		CASE RIFERIMENTO_POSTAZIONE_WA OF
			{Region "CENTRALE" }				
			CENTRALE :
				{Region "ROTAZIONE VERSO 180°" }					  
				IF AngoloRotazioneDestinazionePinza > 95 THEN	
					IF WorkAreaState^[iwa].Supporto.Tipologia = CAVALLETTO THEN 				
						IF (ModuleAX_Y^.Ax^.Status.ActPosition + IngombroDestinazioneY_Pos) >= (QuotaCentroPostazione - WorkAreaState^[iwa].Supporto.YDim/2) AND
							((ModuleAX_Y^.Ax^.Status.ActPosition - IngombroDestinazioneY_Neg) <= QuotaCentroPostazione) OR
							((ModuleAX_Y^.Ax^.Status.ActPosition + IngombroDestinazioneY_Pos) <= (QuotaCentroPostazione - WorkAreaState^[iwa].Supporto.YDim/2)) THEN //Se la pinza è in ingombro con il cavalletto verso SX  
								QuotaFuoriIngombro_Y_Calcolata := MIN(QuotaFuoriIngombro_Y_Calcolata,
																	QuotaCentroPostazione - 						(* Quota Y Postazione *)																									
																	WorkAreaState^[iwa].Supporto.YDim/2 -	(* Dimensione/2 del Pallet/Cassa/Cavallina *)
																	IngombroDestinazioneY_Pos -
																	OffsetSicurezza.Y.Avuoto);
								NuIngombroYCalculado180G_Depuracion := 1;											  
								IF QuotaFuoriIngombro_Y_Calcolata + IngombroDestinazioneY_Pos >= WorkFootprint^[6].Y THEN//Se supero la quota massimo dell'area di lavoro genro un allarme
									Errore := ErrCOLLISIONE_PINZA;
									ErrCollisioneDebug := 110;			 
									RETURN; 
								END_IF
								IF QuotaFuoriIngombro_Y_Calcolata - IngombroDestinazioneY_Neg <= WorkArea^[iwa].Y + INGOMBRO_RISCONTRO_BUNDLE THEN//se sono dentro all'ingombro dei supporti del bundle genero un errore
									Errore := ErrCOLLISIONE_PINZA;
									ErrCollisioneDebug := 111;			 
									RETURN; 
								END_IF			   
						ELSIF (ModuleAX_Y^.Ax^.Status.ActPosition - IngombroDestinazioneY_Neg) >= QuotaCentroPostazione THEN //Se la pinza è in ingombro con il cavalletto  
							QuotaFuoriIngombro_Y_Calcolata := MAX(QuotaFuoriIngombro_Y_Calcolata,
																QuotaCentroPostazione + 						(* Quota Y Postazione *)																									
																WorkAreaState^[iwa].Supporto.YDim/2 +	(* Dimensione/2 del Pallet/Cassa/Cavallina *)
																IngombroDestinazioneY_Neg +
																OffsetSicurezza.Y.Avuoto);
							NuIngombroYCalculado180G_Depuracion := 2;
							IF QuotaFuoriIngombro_Y_Calcolata - IngombroDestinazioneY_Neg <= WorkArea^[iwa].Y + INGOMBRO_RISCONTRO_BUNDLE THEN//se sono dentro all'ingombro dei supporti del bundle genero un errore
								Errore := ErrCOLLISIONE_PINZA;
								ErrCollisioneDebug := 112;
								RETURN;										  
							END_IF											  
							IF QuotaFuoriIngombro_Y_Calcolata + IngombroDestinazioneY_Pos >= WorkFootprint^[6].Y THEN//Se supero la quota massimo dell'area di lavoro genro un allarme
								Errore := ErrCOLLISIONE_PINZA;
								ErrCollisioneDebug := 113;			 
								RETURN; 
							END_IF
						ELSE
							QuotaFuoriIngombro_Y_Calcolata := MAX(QuotaFuoriIngombro_Y_Calcolata,                                                
																QuotaCentroPostazione + 						(* Quota Y Postazione *)				                         																					
																WorkAreaState^[iwa].Supporto.YDim/2 +	(* Dimensione/2 del Pallet/Cassa/Cavallina *)
																IngombroDestinazioneY_Neg +                                                        
																OffsetSicurezza.Y.Avuoto);  
							NuIngombroYCalculado180G_Depuracion := 3;                                                       
							IF QuotaFuoriIngombro_Y_Calcolata - IngombroDestinazioneY_Neg <= WorkArea^[iwa].Y + INGOMBRO_RISCONTRO_BUNDLE THEN//se sono dentro all'ingombro dei supporti del bundle genero un errore
								Errore := ErrCOLLISIONE_PINZA;
								ErrCollisioneDebug := 114;
								RETURN;										  
							END_IF 		
							IF QuotaFuoriIngombro_Y_Calcolata + IngombroDestinazioneY_Pos >= WorkFootprint^[6].Y THEN//Se supero la quota massimo dell'area di lavoro genro un allarme
								Errore := ErrCOLLISIONE_PINZA;
								ErrCollisioneDebug := 115;			 
								RETURN; 
							END_IF																  
						END_IF
					ELSIF WorkAreaState^[iwa].Supporto.Tipologia = BUNDLE THEN //se NELLA postazione c'è un bundle
						IF (ModuleAX_Y^.Ax^.Status.ActPosition - IngombroDestinazioneY_Neg) <= (WorkArea^[iwa].Y + INGOMBRO_RISCONTRO_BUNDLE) THEN //Se la pinza è dentro all'ingombro del bundle  
							QuotaFuoriIngombro_Y_Calcolata := MAX(QuotaFuoriIngombro_Y_Calcolata,
																	QuotaCentroPostazione + 					(* Quota Y Postazione *)																									
																	MAX(WorkAreaState^[iwa].Supporto.YDim,INGOMBRO_RISCONTRO_BUNDLE) + (* massimo tra Dimensione del bundle e dimensione riscontro *)
																	IngombroDestinazioneY_Neg +			(* Ingombro negativo pinza *)
																	OffsetSicurezza.Y.Avuoto);           (* Offset sicurezza *)
							NuIngombroYCalculado180G_Depuracion := 4;
						ELSE
							QuotaFuoriIngombro_Y_Calcolata := MAX(QuotaFuoriIngombro_Y_Calcolata,
																	QuotaCentroPostazione + 					(* Quota Y Postazione *)																									
																	MAX(WorkAreaState^[iwa].Supporto.YDim,INGOMBRO_RISCONTRO_BUNDLE) + (* massimo tra Dimensione del bundle e dimensione riscontro *)
																	IngombroDestinazioneY_Pos +			(* Ingombro negativo pinza *)
																	OffsetSicurezza.Y.Avuoto);           (* Offset sicurezza *)
							NuIngombroYCalculado180G_Depuracion := 5;
						END_IF	
					ELSE//se non c'è nulla o c'è una cassa-pianale
						QuotaFuoriIngombro_Y_Calcolata := MAX(QuotaFuoriIngombro_Y_Calcolata,ModuleAX_Y^.Ax^.Status.ActPosition,WorkSpace^.Y/2 + OffSetPosYReposo);
						IF QuotaFuoriIngombro_Y_Calcolata + IngombroDestinazioneY_Pos >= WorkFootprint^[6].Y THEN//Se supero la quota massima dell'area di lavoro genro un allarme
							Errore := ErrCOLLISIONE_PINZA;
							ErrCollisioneDebug := 116;			 
							RETURN; 
						END_IF	
						IF QuotaFuoriIngombro_Y_Calcolata - IngombroDestinazioneY_Neg <= WorkArea^[iwa].Y + INGOMBRO_RISCONTRO_BUNDLE THEN//se sono dentro all'ingombro dei supporti del bundle genero un errore
							Errore := ErrCOLLISIONE_PINZA;
							ErrCollisioneDebug := 117;			 
							RETURN; 
						END_IF	  
					END_IF
				{endregion}								   
				{Region "ROTAZIONE VERSO 0°" }
				ELSIF AngoloRotazioneDestinazionePinza < 85 THEN
					IF WorkAreaState^[iwa].Supporto.Tipologia = CAVALLETTO THEN 				
						IF (ModuleAX_Y^.Ax^.Status.ActPosition - IngombroDestinazioneY_Neg) <= (QuotaCentroPostazione + WorkAreaState^[iwa].Supporto.YDim/2) AND
						 (ModuleAX_Y^.Ax^.Status.ActPosition - IngombroDestinazioneY_Neg >= QuotaCentroPostazione) OR
						 (ModuleAX_Y^.Ax^.Status.ActPosition - IngombroDestinazioneY_Neg) >= (QuotaCentroPostazione + WorkAreaState^[iwa].Supporto.YDim/2) THEN //Se la pinza è in ingombro con il cavalletto nella zona a SX della sua metà
							QuotaFuoriIngombro_Y_Calcolata := MAX(QuotaFuoriIngombro_Y_Calcolata,
																QuotaCentroPostazione + 						(* Quota Y Postazione *)																									
																WorkAreaState^[iwa].Supporto.YDim/2 +	(* Dimensione/2 del Pallet/Cassa/Cavallina *)
																IngombroDestinazioneY_Neg +
																OffsetSicurezza.Y.Avuoto);
							NuIngombroYCalculado0G_Depuracion := 1;
							IF QuotaFuoriIngombro_Y_Calcolata + IngombroDestinazioneY_Pos >= WorkFootprint^[6].Y THEN//Se supero la quota massimo dell'area di lavoro genro un allarme
								Errore := ErrCOLLISIONE_PINZA;
								ErrCollisioneDebug := 118;			 
								RETURN; 
							END_IF 
						ELSIF ((ModuleAX_Y^.Ax^.Status.ActPosition + IngombroDestinazioneY_Pos) >= (QuotaCentroPostazione - WorkAreaState^[iwa].Supporto.YDim/2) AND 
							(ModuleAX_Y^.Ax^.Status.ActPosition + IngombroDestinazioneY_Pos) <= (QuotaCentroPostazione)) OR
							(ModuleAX_Y^.Ax^.Status.ActPosition + IngombroDestinazioneY_Pos) <= (QuotaCentroPostazione)THEN //Se la pinza è in ingombro con il cavalletto con pinza dentro all'ingombro nella parte SX 
								QuotaFuoriIngombro_Y_Calcolata := MIN(QuotaFuoriIngombro_Y_Calcolata,
																	QuotaCentroPostazione - 						(* Quota Y Postazione *)																									
																	WorkAreaState^[iwa].Supporto.YDim/2 -	(* Dimensione/2 del Pallet/Cassa/Cavallina *)
																	IngombroDestinazioneY_Pos -
																	OffsetSicurezza.Y.Avuoto);
								NuIngombroYCalculado0G_Depuracion := 2;
								IF QuotaFuoriIngombro_Y_Calcolata - IngombroDestinazioneY_Neg <= WorkArea^[iwa].Y + INGOMBRO_RISCONTRO_BUNDLE THEN//se sono dentro all'ingombro dei supporti del bundle genero un errore
									Errore := ErrCOLLISIONE_PINZA;
									ErrCollisioneDebug := 119;
									RETURN;										  
								END_IF 							
						ELSE
							QuotaFuoriIngombro_Y_Calcolata := MAX(QuotaFuoriIngombro_Y_Calcolata,
																QuotaCentroPostazione + 						(* Quota Y Postazione *)																									
																WorkAreaState^[iwa].Supporto.YDim/2 +	(* Dimensione/2 del Pallet/Cassa/Cavallina *)
																IngombroDestinazioneY_Neg +				(* Ingombro positivo pinza *)
																OffsetSicurezza.Y.Avuoto);				(* Offset sicurezza *)
							NuIngombroYCalculado0G_Depuracion := 3;
							IF QuotaFuoriIngombro_Y_Calcolata - IngombroDestinazioneY_Neg <= WorkArea^[iwa].Y + INGOMBRO_RISCONTRO_BUNDLE THEN//se sono dentro all'ingombro dei supporti del bundle genero un errore
								Errore := ErrCOLLISIONE_PINZA;
								ErrCollisioneDebug := 120;
								RETURN;										  
							END_IF 
							IF QuotaFuoriIngombro_Y_Calcolata + IngombroDestinazioneY_Pos >= WorkFootprint^[6].Y THEN//Se supero la quota massimo dell'area di lavoro genro un allarme
								Errore := ErrCOLLISIONE_PINZA;
								ErrCollisioneDebug := 121;			 
								RETURN; 
							END_IF
						END_IF
					ELSIF WorkAreaState^[iwa].Supporto.Tipologia = BUNDLE THEN //se NELLA postazione c'è un bundle
						IF (ModuleAX_Y^.Ax^.Status.ActPosition - IngombroDestinazioneY_Neg) <= (QuotaCentroPostazione + INGOMBRO_RISCONTRO_BUNDLE) THEN //Se la pinza è dentro all'ingombro del bundle  
							QuotaFuoriIngombro_Y_Calcolata := MAX(QuotaFuoriIngombro_Y_Calcolata,
																	QuotaCentroPostazione + 					(* Quota Y Postazione *)																									
																	MAX(WorkAreaState^[iwa].Supporto.YDim,INGOMBRO_RISCONTRO_BUNDLE) + (* massimo tra Dimensione del bundle e dimensione riscontro *)
																	IngombroDestinazioneY_Neg +			(* Ingombro negativo pinza *)
																	OffsetSicurezza.Y.Avuoto);           (* Offset sicurezza *)
							NuIngombroYCalculado0G_Depuracion := 4;
							IF QuotaFuoriIngombro_Y_Calcolata - IngombroDestinazioneY_Neg <= WorkArea^[iwa].Y + INGOMBRO_RISCONTRO_BUNDLE THEN//se sono dentro all'ingombro dei supporti del bundle genero un errore
								Errore := ErrCOLLISIONE_PINZA;
								ErrCollisioneDebug := 122;
								RETURN;										  
							END_IF 
							IF QuotaFuoriIngombro_Y_Calcolata + IngombroDestinazioneY_Pos >= WorkFootprint^[6].Y THEN//Se supero la quota massimo dell'area di lavoro genro un allarme
								Errore := ErrCOLLISIONE_PINZA;
								ErrCollisioneDebug := 123;			 
								RETURN; 
							END_IF												  
						ELSE
							QuotaFuoriIngombro_Y_Calcolata := MAX(QuotaFuoriIngombro_Y_Calcolata,
																	QuotaCentroPostazione + 					(* Quota Y Postazione *)																									
																	MAX(WorkAreaState^[iwa].Supporto.YDim,INGOMBRO_RISCONTRO_BUNDLE) + (* massimo tra Dimensione del bundle e dimensione riscontro *)
																	IngombroDestinazioneY_Pos +			(* Ingombro negativo pinza *)
																	OffsetSicurezza.Y.Avuoto);           (* Offset sicurezza *)
							NuIngombroYCalculado0G_Depuracion := 5;
							IF QuotaFuoriIngombro_Y_Calcolata - IngombroDestinazioneY_Neg <= QuotaCentroPostazione + INGOMBRO_RISCONTRO_BUNDLE THEN//se sono dentro all'ingombro dei supporti del bundle genero un errore
								Errore := ErrCOLLISIONE_PINZA;
								ErrCollisioneDebug := 124;
								RETURN;										  
							END_IF 
							IF QuotaFuoriIngombro_Y_Calcolata + IngombroDestinazioneY_Pos >= WorkFootprint^[6].Y THEN//Se supero la quota massimo dell'area di lavoro genro un allarme
								Errore := ErrCOLLISIONE_PINZA;
								ErrCollisioneDebug := 125;			 
								RETURN; 
							END_IF												  
						END_IF	
					ELSE//se non c'è nulla o c'è una cassa-pianale
						QuotaFuoriIngombro_Y_Calcolata := MAX(QuotaFuoriIngombro_Y_Calcolata,ModuleAX_Y^.Ax^.Status.ActPosition,WorkSpace^.Y/2 +OffSetPosYReposo);
						IF QuotaFuoriIngombro_Y_Calcolata + IngombroDestinazioneY_Pos >= WorkFootprint^[6].Y THEN//Se supero la quota massima dell'area di lavoro genro un allarme
							Errore := ErrCOLLISIONE_PINZA;
							ErrCollisioneDebug := 126;			 
							RETURN; 
						END_IF	
						IF QuotaFuoriIngombro_Y_Calcolata - IngombroDestinazioneY_Neg <= WorkArea^[iwa].Y + INGOMBRO_RISCONTRO_BUNDLE THEN//se sono dentro all'ingombro dei supporti del bundle genero un errore
							Errore := ErrCOLLISIONE_PINZA;
							ErrCollisioneDebug := 127;			 
							RETURN; 
						END_IF	  
					END_IF 	
				{endregion}								   
				{Region "ROTAZIONE 90°" }
				ELSE	
					IF WorkAreaState^[iwa].Supporto.Tipologia = CAVALLETTO THEN 				
						IF (ModuleAX_Y^.Ax^.Status.ActPosition - IngombroDestinazioneY_Neg) <= (QuotaCentroPostazione + WorkAreaState^[iwa].Supporto.YDim/2) AND
							(ModuleAX_Y^.Ax^.Status.ActPosition - IngombroDestinazioneY_Neg >= QuotaCentroPostazione) THEN //Se la pinza è in ingombro con il cavalletto nella zona a DX della sua metà
							QuotaFuoriIngombro_Y_Calcolata := MAX(QuotaFuoriIngombro_Y_Calcolata,
																QuotaCentroPostazione + 						(* Quota Y Postazione *)																									
																WorkAreaState^[iwa].Supporto.YDim/2 +	(* Dimensione/2 del Pallet/Cassa/Cavallina *)
																IngombroDestinazioneY_Neg +
																OffsetSicurezza.Y.Avuoto);
						NuIngombroYCalculado90G_Depuracion := 1 ;
							IF QuotaFuoriIngombro_Y_Calcolata + IngombroDestinazioneY_Pos >= WorkFootprint^[6].Y THEN//Se supero la quota massimo dell'area di lavoro genro un allarme
								Errore := ErrCOLLISIONE_PINZA;
								ErrCollisioneDebug := 128;			 
								RETURN; 
							END_IF 
						ELSIF (ModuleAX_Y^.Ax^.Status.ActPosition + IngombroDestinazioneY_Pos) >= (QuotaCentroPostazione - WorkAreaState^[iwa].Supporto.YDim/2) AND 
							(ModuleAX_Y^.Ax^.Status.ActPosition + IngombroDestinazioneY_Pos) <= (QuotaCentroPostazione) THEN //Se la pinza è in ingombro con il cavalletto con pinza dentro all'ingombro nella parte SX 
								QuotaFuoriIngombro_Y_Calcolata := MIN(QuotaFuoriIngombro_Y_Calcolata,
																	QuotaCentroPostazione - 						(* Quota Y Postazione *)																									
																	WorkAreaState^[iwa].Supporto.YDim/2 -	(* Dimensione/2 del Pallet/Cassa/Cavallina *)
																	IngombroDestinazioneY_Pos -
																	OffsetSicurezza.Y.Avuoto);
							NuIngombroYCalculado90G_Depuracion := 2 ;
								IF QuotaFuoriIngombro_Y_Calcolata - IngombroDestinazioneY_Neg <= WorkArea^[iwa].Y + INGOMBRO_RISCONTRO_BUNDLE THEN//se sono dentro all'ingombro dei supporti del bundle genero un errore
									Errore := ErrCOLLISIONE_PINZA;
									ErrCollisioneDebug := 129;
									RETURN;										  
								END_IF 							
						ELSE
							QuotaFuoriIngombro_Y_Calcolata := MAX(QuotaFuoriIngombro_Y_Calcolata,
																QuotaCentroPostazione + 						(* Quota Y Postazione *)																									
																WorkAreaState^[iwa].Supporto.YDim/2 +	(* Dimensione/2 del Pallet/Cassa/Cavallina *)
																IngombroDestinazioneY_Neg +				(* Ingombro positivo pinza *)
																OffsetSicurezza.Y.Avuoto);				(* Offset sicurezza *)
							NuIngombroYCalculado90G_Depuracion := 3 ;
							IF QuotaFuoriIngombro_Y_Calcolata - IngombroDestinazioneY_Neg <= WorkArea^[iwa].Y + INGOMBRO_RISCONTRO_BUNDLE THEN//se sono dentro all'ingombro dei supporti del bundle genero un errore
								Errore := ErrCOLLISIONE_PINZA;
								ErrCollisioneDebug := 130;
								RETURN;										  
							END_IF 
							IF QuotaFuoriIngombro_Y_Calcolata + IngombroDestinazioneY_Pos >= WorkFootprint^[6].Y THEN//Se supero la quota massimo dell'area di lavoro genro un allarme
								Errore := ErrCOLLISIONE_PINZA;
								ErrCollisioneDebug := 131;			 
								RETURN; 
							END_IF
						END_IF
					ELSIF WorkAreaState^[iwa].Supporto.Tipologia = BUNDLE THEN //se NELLA postazione c'è un bundle
						IF (ModuleAX_Y^.Ax^.Status.ActPosition - IngombroDestinazioneY_Neg) <= (WorkArea^[iwa].Y + INGOMBRO_RISCONTRO_BUNDLE) THEN //Se la pinza è dentro all'ingombro del bundle  
							QuotaFuoriIngombro_Y_Calcolata := MAX(QuotaFuoriIngombro_Y_Calcolata,
																	QuotaCentroPostazione + 					(* Quota Y Postazione *)																									
																	MAX(WorkAreaState^[iwa].Supporto.YDim,INGOMBRO_RISCONTRO_BUNDLE) + (* massimo tra Dimensione del bundle e dimensione riscontro *)
																	IngombroDestinazioneY_Neg +			(* Ingombro negativo pinza *)
																	OffsetSicurezza.Y.Avuoto);           (* Offset sicurezza *)
							NuIngombroYCalculado90G_Depuracion := 4 ;
							IF QuotaFuoriIngombro_Y_Calcolata - IngombroDestinazioneY_Neg <= WorkArea^[iwa].Y + INGOMBRO_RISCONTRO_BUNDLE THEN//se sono dentro all'ingombro dei supporti del bundle genero un errore
								Errore := ErrCOLLISIONE_PINZA;
								ErrCollisioneDebug := 132;
								RETURN;										  
							END_IF 
							IF QuotaFuoriIngombro_Y_Calcolata + IngombroDestinazioneY_Pos >= WorkFootprint^[6].Y THEN//Se supero la quota massimo dell'area di lavoro genro un allarme
								Errore := ErrCOLLISIONE_PINZA;
								ErrCollisioneDebug := 133;			 
								RETURN; 
							END_IF												  
						ELSE
							QuotaFuoriIngombro_Y_Calcolata := MAX(QuotaFuoriIngombro_Y_Calcolata,
																	QuotaCentroPostazione + 					(* Quota Y Postazione *)																									
																	MAX(WorkAreaState^[iwa].Supporto.YDim,INGOMBRO_RISCONTRO_BUNDLE) + (* massimo tra Dimensione del bundle e dimensione riscontro *)
																	IngombroDestinazioneY_Pos +			(* Ingombro negativo pinza *)
																	OffsetSicurezza.Y.Avuoto);           (* Offset sicurezza *)
							NuIngombroYCalculado90G_Depuracion := 5 ;
							IF QuotaFuoriIngombro_Y_Calcolata - IngombroDestinazioneY_Neg <= WorkArea^[iwa].Y + INGOMBRO_RISCONTRO_BUNDLE THEN//se sono dentro all'ingombro dei supporti del bundle genero un errore
								Errore := ErrCOLLISIONE_PINZA;
								ErrCollisioneDebug := 134;
								RETURN;										  
							END_IF 
							IF QuotaFuoriIngombro_Y_Calcolata + IngombroDestinazioneY_Pos >= WorkFootprint^[6].Y THEN//Se supero la quota massimo dell'area di lavoro genro un allarme
								Errore := ErrCOLLISIONE_PINZA;
								ErrCollisioneDebug := 135;			 
								RETURN; 
							END_IF												  
						END_IF	
					ELSE//se non c'è nulla o c'è una cassa-pianale
						QuotaFuoriIngombro_Y_Calcolata := MAX(QuotaFuoriIngombro_Y_Calcolata,ModuleAX_Y^.Ax^.Status.ActPosition,WorkSpace^.Y/2+ OffSetPosYReposo);
						IF QuotaFuoriIngombro_Y_Calcolata + IngombroDestinazioneY_Pos >= WorkFootprint^[6].Y THEN//Se supero la quota massima dell'area di lavoro genro un allarme
							Errore := ErrCOLLISIONE_PINZA;
							ErrCollisioneDebug := 136;			 
							RETURN; 
						END_IF	
						IF QuotaFuoriIngombro_Y_Calcolata - IngombroDestinazioneY_Neg <= WorkArea^[iwa].Y + INGOMBRO_RISCONTRO_BUNDLE THEN//se sono dentro all'ingombro dei supporti del bundle genero un errore
							Errore := ErrCOLLISIONE_PINZA;
							ErrCollisioneDebug := 137;			 
							RETURN; 
						END_IF	  
					END_IF
				END_IF
				{endregion}				   
			{endregion}
		
		ELSE
			;//Errore.Code := ErrWAM_FTC_PostazioneNONDefinita;
		END_CASE
	{endregion}	
	{region " Pallettizzatore SX "}	
	PALLETTIZZATORE_SX:
		CASE RIFERIMENTO_POSTAZIONE_WA OF
		{Region "CENTRALE" }				
			CENTRALE :
				{Region "ROTAZIONE VERSO 180°" }					  
				IF AngoloRotazioneDestinazionePinza > 95 THEN
					//Modificacar aqui para salir <cavaleta	
					IF WorkAreaState^[iwa].Supporto.Tipologia = CAVALLETTO  (*Añadido*)OR WorkAreaState^[PosRobot].Supporto.Tipologia = CAVALLETTO 
							OR (WorkAreaState^[Mission^.PPlace].Supporto.Tipologia = CAVALLETTO	AND WorkAreaManager^.State = 	WAMANAGER_CICLO_DEPOSITO_LASTRA_WA_RUN)	THEN 				
						IF (ModuleAX_Y^.Ax^.Status.ActPosition + IngombroDestinazioneY_Pos) >= (QuotaCentroPostazione - WorkAreaState^[iwa].Supporto.YDim/2) AND
							((ModuleAX_Y^.Ax^.Status.ActPosition - IngombroDestinazioneY_Neg) <= QuotaCentroPostazione) OR
							((ModuleAX_Y^.Ax^.Status.ActPosition + IngombroDestinazioneY_Pos) <= (QuotaCentroPostazione - WorkAreaState^[iwa].Supporto.YDim/2)) OR
							 	( (WorkAreaState^[PosRobot].Supporto.Tipologia = CAVALLETTO OR WorkAreaState^[Mission^.PPlace].Supporto.Tipologia = CAVALLETTO ) AND ModuleAX_Y^.Ax^.Status.ActPosition + IngombroDestinazioneY_Pos < WorkFootprint^[6].Y )THEN //Se la pinza è in ingombro con il cavalletto verso SX  
							 	IF WorkAreaState^[PosRobot].Supporto.Tipologia = CAVALLETTO OR  
											WorkAreaState^[Mission^.PPlace].Supporto.Tipologia = CAVALLETTO THEN
									IF WorkAreaState^[Mission^.PPlace].Supporto.Tipologia = CAVALLETTO AND WorkAreaManager^.State = 	WAMANAGER_CICLO_DEPOSITO_LASTRA_WA_RUN  THEN
											QuotaFuoriIngombro_Y_Calcolata := 
													   //%%%%%%%%%%%%%%%%modificado 18-7-2025
																			MAX(QuotaFuoriIngombro_Y_Calcolata,
																			QuotaCentroPostazionePiking + 						(* Quota Y Postazione *)																									
																			WorkAreaState^[Mission^.PPlace].Supporto.YDim/2 (*-	        (* Dimensione/2 del Pallet/Cassa/Cavallina *)
																			IngombroDestinazioneY_Pos - *) 
																			+ Max (OffsetSicurezza.Y.Avuoto ,Dimensioni_Pinza.Spessore)           )  ;
									NuIngombroYCalculado180G_Depuracion := 6;
									ELSE
										IF Mission^.PPick = PosRobot AND( Mission^.JPick <> Mission^.JPlace OR ModuleAX_J^.Ax^.Status.ActPosition < 85) THEN
														   
											IF 	Mission^.JPick < 85 THEN
											QuotaFuoriIngombro_Y_Calcolata := 
											 //%%%%%%%%%%%%%%%%modificado 18-7-2025
																			MAX(QuotaFuoriIngombro_Y_Calcolata,
																			QuotaCentroPostazioneIni - 						(* Quota Y Postazione *)																									
																			WorkAreaState^[Mission^.PPick].Supporto.YDim/2 (*-	        (* Dimensione/2 del Pallet/Cassa/Cavallina *)
																			IngombroDestinazioneY_Pos - *) 
																			- OffsetSicurezza.Y.Avuoto )  ;	
											NuIngombroYCalculado180G_Depuracion := 7;	   
	   										ELSE
											QuotaFuoriIngombro_Y_Calcolata := 
											 //%%%%%%%%%%%%%%%%modificado 18-7-2025
																			MAX(QuotaFuoriIngombro_Y_Calcolata,
																			QuotaCentroPostazioneIni + 						(* Quota Y Postazione *)																									
																			WorkAreaState^[Mission^.PPick].Supporto.YDim/2 (*-	        (* Dimensione/2 del Pallet/Cassa/Cavallina *)
																			IngombroDestinazioneY_Pos - *) 
																			+ OffsetSicurezza.Y.Avuoto )  ;	
											NuIngombroYCalculado180G_Depuracion := 8;	   				   
											END_IF	
										// Añadido 	29 -7-2025__________________________________________			   
										ELSIF   PosRobot <> 0 AND   WorkAreaState^[PosRobot].Supporto.Tipologia = CAVALLETTO  AND ModuleAX_J^.Ax^.Status.ActPosition > 95      THEN 
											QuotaFuoriIngombro_Y_Calcolata := 
											 //%%%%%%%%%%%%%%%%modificado 18-7-2025
																			MAX(QuotaFuoriIngombro_Y_Calcolata,
																			QuotaCentroPostazioneIni  + 						(* Quota Y Postazione *)	
																			//	WorkAreaState^[Mission^.PPick].Supporto.YDim/2				
																			WorkAreaState^[PosRobot].Supporto.YDim /2 (*-	        (* Dimensione/2 del Pallet/Cassa/Cavallina *)
																			
																			IngombroDestinazioneY_Pos - *) 
																			+ OffsetSicurezza.Y.Avuoto +INGOMBRO_RISCONTRO_FRAME )  ;
										NuIngombroYCalculado180G_Depuracion := 9;			   			   
		   								// Añadido 	29 -7-2025_________________________________________________
										ELSIF PosRobot <> 0 AND  WorkAreaState^[PosRobot].Supporto.Tipologia = CAVALLETTO  AND ModuleAX_J^.Ax^.Status.ActPosition < 95    THEN 
											
																			
																			IF 	WorkAreaState^[Mission^.PPick].Supporto.Tipologia = BUNDLE THEN
																				Soporte := WorkAreaState^[Mission^.PPick].Supporto.YDim;	
																			ELSIF WorkAreaState^[Mission^.PPick].Supporto.Tipologia = CAVALLETTO THEN
																				Soporte := WorkAreaState^[Mission^.PPick].Supporto.YDim /2;	   
																			END_IF		   
																			QuotaFuoriIngombro_Y_Calcolata := 
																			 //%%%%%%%%%%%%%%%%modificado 18-7-2025														  
																			//Modificacion Pasillo Trabajo Caballete
																			MAX(QuotaFuoriIngombro_Y_Calcolata,
																			QuotaCentroPostazione  + 					(* Quota Y Postazione *)	
																			Soporte
																			+ MAX( OffsetSicurezza.Y.Avuoto , Dimensioni_Pinza.Spessore))  ;
										NuIngombroYCalculado180G_Depuracion := 10;		   			   
		   								// Añadido 	2 -9-2025_________________________________________________
										ELSIF (( WorkAreaState^[Mission^.PPick].Supporto.Tipologia = CAVALLETTO  AND NuPosGuiroPiking = PosRobot) OR ( PosRobot <> 0 AND WorkAreaState^[PosRobot].Supporto.Tipologia <> CAVALLETTO))  AND PosicionJActual = 90     THEN 
											QuotaFuoriIngombro_Y_Calcolata := 
											 //%%%%%%%%%%%%%%%%modificado 2-9-2025
																			MAX(QuotaFuoriIngombro_Y_Calcolata,
																			QuotaCentroPostazione  + 						(* Quota Y Postazione *)	
																			//	WorkAreaState^[Mission^.PPick].Supporto.YDim/2				
																			WorkAreaState^[Mission^.PPick].Supporto.YDim /2 + Dimensioni_Pinza.Spessore(*-	        (* Dimensione/2 del Pallet/Cassa/Cavallina *)
																			
																			IngombroDestinazioneY_Pos - *) 
																			(*+ OffsetSicurezza.Y.Avuoto *)+ INGOMBRO_RISCONTRO_FRAME)  ;	
										NuIngombroYCalculado180G_Depuracion := 11;		
										// Añadido 	4 -9-2025_________________________________________________
										ELSIF  WorkAreaState^[Mission^.PPick].Supporto.Tipologia = BUNDLE  AND  PosRobot = 0    THEN 
											QuotaFuoriIngombro_Y_Calcolata := 
											 //%%%%%%%%%%%%%%%%modificado 2-9-2025
																			MAX(QuotaFuoriIngombro_Y_Calcolata,
																			QuotaCentroPostazione  + 						(* Quota Y Postazione *)	
																			//	WorkAreaState^[Mission^.PPick].Supporto.YDim/2				
																			WorkAreaState^[Mission^.PPick].Supporto.YDim /2 (*-	        (* Dimensione/2 del Pallet/Cassa/Cavallina *)
																			
																			IngombroDestinazioneY_Pos - *) 
																			+ OffsetSicurezza.Y.Avuoto )  ;		
										NuIngombroYCalculado180G_Depuracion := 12;	   		   			
										END_IF
										 
									END_IF
								ELSE
										IF 	WorkAreaState^[Mission^.PPlace].Supporto.Tipologia = CAVALLETTO	 THEN
  											QuotaFuoriIngombro_Y_Calcolata := 
											   //%%%%%%%%%%%%%%%%modificado 18-7-2025
											   						MAX(QuotaFuoriIngombro_Y_Calcolata,
																	QuotaCentroPostazione + 						(* Quota Y Postazione *)																									
																	WorkAreaState^[iwa].Supporto.YDim/2 (*-	        (* Dimensione/2 del Pallet/Cassa/Cavallina *)
																	IngombroDestinazioneY_Pos - *) 
																	+ OffsetSicurezza.Y.Avuoto + INGOMBRO_RISCONTRO_FRAME )  ;
										NuIngombroYCalculado180G_Depuracion := 13;
										ELSIF WorkAreaState^[Mission^.PPlace].Supporto.Tipologia = BUNDLE    THEN  	
											QuotaFuoriIngombro_Y_Calcolata := 
											   //%%%%%%%%%%%%%%%%modificado 18-7-2025
											   						MAX(QuotaFuoriIngombro_Y_Calcolata,
																	QuotaCentroPostazione + 						(* Quota Y Postazione *)																									
																	WorkAreaState^[iwa].Supporto.YDim /2  (*-	        (* Dimensione/2 del Pallet/Cassa/Cavallina *)
																	IngombroDestinazioneY_Pos - *) 
																	+MAX(Dimensioni_Pinza.Spessore ,OffsetSicurezza.Y.Avuoto ))+ INGOMBRO_RISCONTRO_FRAME   ;
										NuIngombroYCalculado180G_Depuracion := 14;
											ELSIF WorkAreaState^[Mission^.PPick].Supporto.Tipologia = CAVALLETTO    THEN  	
											QuotaFuoriIngombro_Y_Calcolata := 
											   //%%%%%%%%%%%%%%%%modificado 18-7-2025
											   						MAX(QuotaFuoriIngombro_Y_Calcolata,
																	QuotaCentroPostazione + 						(* Quota Y Postazione *)																									
																	WorkAreaState^[iwa].Supporto.YDim /2 (*-	        (* Dimensione/2 del Pallet/Cassa/Cavallina *)
																	IngombroDestinazioneY_Pos - *) 
																	+ max ( Dimensioni_Pinza.Spessore ,  OffsetSicurezza.Y.Avuoto )+ INGOMBRO_RISCONTRO_FRAME )  ;	
										NuIngombroYCalculado180G_Depuracion := 15;							
										END_IF 
					  
			   						
								END_IF 		   
										(*	QuotaFuoriIngombro_Y_Calcolata := 
											   //%%%%%%%%%%%%%%%%modificado 18-7-2025
											   						MAX(QuotaFuoriIngombro_Y_Calcolata,
																	QuotaCentroPostazione + 						(* Quota Y Postazione *)																									
																	WorkAreaState^[iwa].Supporto.YDim/2 (*-	        (* Dimensione/2 del Pallet/Cassa/Cavallina *)
																	IngombroDestinazioneY_Pos - *) 
																	+ OffsetSicurezza.Y.Avuoto )  ;
																(*	MIN(QuotaFuoriIngombro_Y_Calcolata,
																	QuotaCentroPostazione - 						(* Quota Y Postazione *)																									
																	WorkAreaState^[iwa].Supporto.YDim/2 -	(* Dimensione/2 del Pallet/Cassa/Cavallina *)
																	IngombroDestinazioneY_Pos -
																	OffsetSicurezza.Y.Avuoto);*)
																			  *)
								IF QuotaFuoriIngombro_Y_Calcolata (*+ IngombroDestinazioneY_Pos*) >= WorkFootprint^[6].Y THEN//Se supero la quota massimo dell'area di lavoro genro un allarme
									Errore := ErrCOLLISIONE_PINZA;
									ErrCollisioneDebug := 10;			 
									RETURN; 
								END_IF
								IF QuotaFuoriIngombro_Y_Calcolata - IngombroDestinazioneY_Neg <= WorkArea^[iwa].Y + INGOMBRO_RISCONTRO_BUNDLE THEN//se sono dentro all'ingombro dei supporti del bundle genero un errore
									Errore := ErrCOLLISIONE_PINZA;
									ErrCollisioneDebug := 11;			 
									RETURN; 
								END_IF			   
						ELSIF (ModuleAX_Y^.Ax^.Status.ActPosition - IngombroDestinazioneY_Neg) >= QuotaCentroPostazione THEN //Se la pinza è in ingombro con il cavalletto  
							QuotaFuoriIngombro_Y_Calcolata := MAX(QuotaFuoriIngombro_Y_Calcolata,
																QuotaCentroPostazione + 						(* Quota Y Postazione *)																									
																WorkAreaState^[iwa].Supporto.YDim/2 +	(* Dimensione/2 del Pallet/Cassa/Cavallina *)
																IngombroDestinazioneY_Neg + INGOMBRO_RISCONTRO_FRAME(*+
																OffsetSicurezza.Y.Avuoto*));
							NuIngombroYCalculado180G_Depuracion := 16;
							IF QuotaFuoriIngombro_Y_Calcolata - IngombroDestinazioneY_Neg <= WorkArea^[iwa].Y + INGOMBRO_RISCONTRO_BUNDLE THEN//se sono dentro all'ingombro dei supporti del bundle genero un errore
								Errore := ErrCOLLISIONE_PINZA;
								ErrCollisioneDebug := 12;
								RETURN;										  
							END_IF											  
							IF QuotaFuoriIngombro_Y_Calcolata + IngombroDestinazioneY_Pos /2(*Puesto Para Probar*)  >= WorkFootprint^[6].Y THEN//Se supero la quota massimo dell'area di lavoro genro un allarme
								Errore := ErrCOLLISIONE_PINZA;
								ErrCollisioneDebug := 13;			 
								RETURN; 
							END_IF
						ELSE
							QuotaFuoriIngombro_Y_Calcolata := MAX(QuotaFuoriIngombro_Y_Calcolata,                                                
																QuotaCentroPostazione + 						(* Quota Y Postazione *)				                         																					
																WorkAreaState^[iwa].Supporto.YDim/2 +	(* Dimensione/2 del Pallet/Cassa/Cavallina *)
																(*IngombroDestinazioneY_Neg + *) //+++++++++                                                      
																OffsetSicurezza.Y.Avuoto);  
							NuIngombroYCalculado180G_Depuracion := 17;                                                       
							IF QuotaFuoriIngombro_Y_Calcolata - IngombroDestinazioneY_Neg <= WorkArea^[iwa].Y + INGOMBRO_RISCONTRO_BUNDLE THEN//se sono dentro all'ingombro dei supporti del bundle genero un errore
								Errore := ErrCOLLISIONE_PINZA;
								ErrCollisioneDebug := 14;
								RETURN;										  
							END_IF 		
							IF QuotaFuoriIngombro_Y_Calcolata + IngombroDestinazioneY_Pos >= WorkFootprint^[6].Y THEN//Se supero la quota massimo dell'area di lavoro genro un allarme
								Errore := ErrCOLLISIONE_PINZA;
								ErrCollisioneDebug := 15;			 
								RETURN; 
							END_IF																  
						END_IF
					ELSIF WorkAreaState^[iwa].Supporto.Tipologia = BUNDLE THEN //se NELLA postazione c'è un bundle
						IF (ModuleAX_Y^.Ax^.Status.ActPosition - IngombroDestinazioneY_Neg) <= (WorkArea^[iwa].Y + INGOMBRO_RISCONTRO_BUNDLE) THEN //Se la pinza è dentro all'ingombro del bundle  
							QuotaFuoriIngombro_Y_Calcolata := MAX(QuotaFuoriIngombro_Y_Calcolata,
																	QuotaCentroPostazione + 					(* Quota Y Postazione *)																									
																	MAX(WorkAreaState^[iwa].Supporto.YDim,INGOMBRO_RISCONTRO_BUNDLE) + (* massimo tra Dimensione del bundle e dimensione riscontro *)
																	MAX (IngombroDestinazioneY_Neg ,			(* Ingombro negativo pinza *)
																	OffsetSicurezza.Y.Avuoto));           (* Offset sicurezza *)
						NuIngombroYCalculado180G_Depuracion := 18; 
						ELSE
							QuotaFuoriIngombro_Y_Calcolata := MAX(QuotaFuoriIngombro_Y_Calcolata,
																	QuotaCentroPostazione + 					(* Quota Y Postazione *)																									
																	MAX(WorkAreaState^[iwa].Supporto.YDim,INGOMBRO_RISCONTRO_BUNDLE) + (* massimo tra Dimensione del bundle e dimensione riscontro *)
																	MAX (IngombroDestinazioneY_Pos  ,			(* Ingombro negativo pinza *)
																	OffsetSicurezza.Y.Avuoto, Dimensioni_Pinza.Spessore) +INGOMBRO_RISCONTRO_BUNDLE);           (* Offset sicurezza *)
						NuIngombroYCalculado180G_Depuracion := 19; 
						END_IF	
					ELSE//se non c'è nulla o c'è una cassa-pianale
						QuotaFuoriIngombro_Y_Calcolata := MAX(QuotaFuoriIngombro_Y_Calcolata,ModuleAX_Y^.Ax^.Status.ActPosition,WorkSpace^.Y/2 + OffSetPosYReposo);
						IF QuotaFuoriIngombro_Y_Calcolata + IngombroDestinazioneY_Pos >= WorkFootprint^[6].Y THEN//Se supero la quota massima dell'area di lavoro genro un allarme
							Errore := ErrCOLLISIONE_PINZA;
							ErrCollisioneDebug := 16;			 
							RETURN; 
						END_IF	
						IF QuotaFuoriIngombro_Y_Calcolata - IngombroDestinazioneY_Neg <= WorkArea^[iwa].Y + INGOMBRO_RISCONTRO_BUNDLE THEN//se sono dentro all'ingombro dei supporti del bundle genero un errore
							Errore := ErrCOLLISIONE_PINZA;
							ErrCollisioneDebug := 17;			 
							RETURN; 
						END_IF	  
					END_IF
				{endregion}								   
				{Region "ROTAZIONE VERSO 0°" }
				ELSIF AngoloRotazioneDestinazionePinza < 85 THEN
					IF WorkAreaState^[iwa].Supporto.Tipologia = CAVALLETTO THEN 				
						IF (ModuleAX_Y^.Ax^.Status.ActPosition - IngombroDestinazioneY_Neg) <= (QuotaCentroPostazione + WorkAreaState^[iwa].Supporto.YDim/2) AND
							(ModuleAX_Y^.Ax^.Status.ActPosition - IngombroDestinazioneY_Neg >= QuotaCentroPostazione) THEN //Se la pinza è in ingombro con il cavalletto nella zona a DX della sua metà
							QuotaFuoriIngombro_Y_Calcolata := MAX(QuotaFuoriIngombro_Y_Calcolata,
																QuotaCentroPostazione - 						(* Quota Y Postazione *)																									
																WorkAreaState^[iwa].Supporto.YDim/2 -	(* Dimensione/2 del Pallet/Cassa/Cavallina *)
																IngombroDestinazioneY_Neg  -
																OffsetSicurezza.Y.Avuoto );
						   NuIngombroYCalculado0G_Depuracion := 6;	
							(*												   
							QuotaFuoriIngombro_Y_Calcolata := MAX(QuotaFuoriIngombro_Y_Calcolata,
																QuotaCentroPostazione + 						(* Quota Y Postazione *)																									
																WorkAreaState^[iwa].Supporto.YDim/2 +	(* Dimensione/2 del Pallet/Cassa/Cavallina *)
																IngombroDestinazioneY_Neg +
																OffsetSicurezza.Y.Avuoto);												   
								*)
							IF QuotaFuoriIngombro_Y_Calcolata + IngombroDestinazioneY_Pos >= WorkFootprint^[6].Y THEN//Se supero la quota massimo dell'area di lavoro genro un allarme
								Errore := ErrCOLLISIONE_PINZA;
								ErrCollisioneDebug := 18;			 
								RETURN; 
							END_IF 
						ELSIF (ModuleAX_Y^.Ax^.Status.ActPosition + IngombroDestinazioneY_Pos) >= (QuotaCentroPostazione - WorkAreaState^[iwa].Supporto.YDim/2) AND 
							(ModuleAX_Y^.Ax^.Status.ActPosition + IngombroDestinazioneY_Pos <= QuotaCentroPostazione) THEN //Se la pinza è in ingombro con il cavalletto con pinza dentro all'ingombro nella parte SX 
								QuotaFuoriIngombro_Y_Calcolata := //MIN(QuotaFuoriIngombro_Y_Calcolata,
												   				   MAX(QuotaFuoriIngombro_Y_Calcolata,
																	QuotaCentroPostazione - 						(* Quota Y Postazione *)																									
																	WorkAreaState^[iwa].Supporto.YDim/2 -	(* Dimensione/2 del Pallet/Cassa/Cavallina *)
																	MAX( IngombroDestinazioneY_Pos ,
																	OffsetSicurezza.Y.Avuoto));
							   NuIngombroYCalculado0G_Depuracion := 7;
								IF QuotaFuoriIngombro_Y_Calcolata - IngombroDestinazioneY_Neg <= WorkArea^[iwa].Y + INGOMBRO_RISCONTRO_BUNDLE THEN//se sono dentro all'ingombro dei supporti del bundle genero un errore
									Errore := ErrCOLLISIONE_PINZA;
									ErrCollisioneDebug := 19;
									RETURN;										  
								END_IF 							
						ELSE
							QuotaFuoriIngombro_Y_Calcolata := MAX(QuotaFuoriIngombro_Y_Calcolata,
																QuotaCentroPostazione - 						(* Quota Y Postazione *)																									
																WorkAreaState^[iwa].Supporto.YDim/2 -	(* Dimensione/2 del Pallet/Cassa/Cavallina *)
																IngombroDestinazioneY_Neg -				(* Ingombro positivo pinza *)
																MAX( IngombroDestinazioneY_Pos ,
																	OffsetSicurezza.Y.Avuoto));				(* Offset sicurezza *)
						   NuIngombroYCalculado0G_Depuracion := 8;
															(*	
																QuotaCentroPostazione + 						(* Quota Y Postazione *)																									
																WorkAreaState^[iwa].Supporto.YDim/2 +	(* Dimensione/2 del Pallet/Cassa/Cavallina *)
																IngombroDestinazioneY_Neg +				(* Ingombro positivo pinza *)
																OffsetSicurezza.Y.Avuoto);				(* Offset sicurezza *)
																			   *)
							IF QuotaFuoriIngombro_Y_Calcolata - IngombroDestinazioneY_Neg <= WorkArea^[iwa].Y + INGOMBRO_RISCONTRO_BUNDLE THEN//se sono dentro all'ingombro dei supporti del bundle genero un errore
								Errore := ErrCOLLISIONE_PINZA;
								ErrCollisioneDebug := 20;
								RETURN;										  
							END_IF 
							IF QuotaFuoriIngombro_Y_Calcolata + IngombroDestinazioneY_Pos >= WorkFootprint^[6].Y THEN//Se supero la quota massimo dell'area di lavoro genro un allarme
								Errore := ErrCOLLISIONE_PINZA;
								ErrCollisioneDebug := 21;			 
								RETURN; 
							END_IF
						END_IF
					ELSIF WorkAreaState^[iwa].Supporto.Tipologia = BUNDLE THEN //se NELLA postazione c'è un bundle
						IF (ModuleAX_Y^.Ax^.Status.ActPosition - IngombroDestinazioneY_Neg) <= (QuotaCentroPostazione + INGOMBRO_RISCONTRO_BUNDLE) THEN //Se la pinza è dentro all'ingombro del bundle  
							QuotaFuoriIngombro_Y_Calcolata := MAX(QuotaFuoriIngombro_Y_Calcolata,
																	QuotaCentroPostazione + 					(* Quota Y Postazione *)																									
																	MAX(WorkAreaState^[iwa].Supporto.YDim,INGOMBRO_RISCONTRO_BUNDLE) + (* massimo tra Dimensione del bundle e dimensione riscontro *)
																	IngombroDestinazioneY_Neg +			(* Ingombro negativo pinza *)
																	OffsetSicurezza.Y.Avuoto);           (* Offset sicurezza *)
						   NuIngombroYCalculado0G_Depuracion := 9;
							IF QuotaFuoriIngombro_Y_Calcolata - IngombroDestinazioneY_Neg <= WorkArea^[iwa].Y + INGOMBRO_RISCONTRO_BUNDLE THEN//se sono dentro all'ingombro dei supporti del bundle genero un errore
								Errore := ErrCOLLISIONE_PINZA;
								ErrCollisioneDebug := 22;
								RETURN;										  
							END_IF 
							IF QuotaFuoriIngombro_Y_Calcolata + IngombroDestinazioneY_Pos >= WorkFootprint^[6].Y THEN//Se supero la quota massimo dell'area di lavoro genro un allarme
								Errore := ErrCOLLISIONE_PINZA;
								ErrCollisioneDebug := 23;			 
								RETURN; 
							END_IF												  
						ELSE
							QuotaFuoriIngombro_Y_Calcolata := MAX(QuotaFuoriIngombro_Y_Calcolata,
																	QuotaCentroPostazione + 					(* Quota Y Postazione *)																									
																	MAX(WorkAreaState^[iwa].Supporto.YDim,INGOMBRO_RISCONTRO_BUNDLE) + (* massimo tra Dimensione del bundle e dimensione riscontro *)
																	IngombroDestinazioneY_Pos +			(* Ingombro negativo pinza *)
																	OffsetSicurezza.Y.Avuoto);           (* Offset sicurezza *)
						   NuIngombroYCalculado0G_Depuracion := 10;
							IF QuotaFuoriIngombro_Y_Calcolata - IngombroDestinazioneY_Neg <= WorkArea^[iwa].Y + INGOMBRO_RISCONTRO_BUNDLE THEN//se sono dentro all'ingombro dei supporti del bundle genero un errore
								Errore := ErrCOLLISIONE_PINZA;
								ErrCollisioneDebug := 24;
								RETURN;										  
							END_IF 
							IF QuotaFuoriIngombro_Y_Calcolata + IngombroDestinazioneY_Pos >= WorkFootprint^[6].Y THEN//Se supero la quota massimo dell'area di lavoro genro un allarme
								Errore := ErrCOLLISIONE_PINZA;
								ErrCollisioneDebug := 25;			 
								RETURN; 
							END_IF												  
						END_IF	
					ELSE//se non c'è nulla o c'è una cassa-pianale
						QuotaFuoriIngombro_Y_Calcolata :=  
															(*MAX(QuotaFuoriIngombro_Y_Calcolata,
										   						WorkArea^[iwa].Y + INGOMBRO_RISCONTRO_BUNDLE,//comunque devo sempre considerarlo perchè il riscontro è sempre presente!!!!
																//ModuleAX_Y^.Ax^.Status.ActPosition,WorkSpace^.Y/2+ OffSetPosYReposo);		   
																ModuleAX_Y^.Ax^.Status.ActPosition,WorkSpace^.Y/2(*+ OffSetPosYReposo*)); *)
															MIN(QuotaFuoriIngombro_Y_Calcolata,
										   						MAX(WorkArea^[iwa].Y + INGOMBRO_RISCONTRO_BUNDLE,//comunque devo sempre considerarlo perchè il riscontro è sempre presente!!!!
																//ModuleAX_Y^.Ax^.Status.ActPosition,WorkSpace^.Y/2+ OffSetPosYReposo);		   
																ModuleAX_Y^.Ax^.Status.ActPosition,WorkSpace^.Y/2(*+ OffSetPosYReposo*)));	
						NuIngombroYCalculado0G_Depuracion := 11;			   
																							  
						IF QuotaFuoriIngombro_Y_Calcolata + IngombroDestinazioneY_Pos >= WorkFootprint^[6].Y THEN//Se supero la quota massima dell'area di lavoro genro un allarme
							Errore := ErrCOLLISIONE_PINZA;
							ErrCollisioneDebug := 26;			 
							RETURN; 
						END_IF	
						IF QuotaFuoriIngombro_Y_Calcolata - IngombroDestinazioneY_Neg <= WorkArea^[iwa].Y + INGOMBRO_RISCONTRO_BUNDLE THEN//se sono dentro all'ingombro dei supporti del bundle genero un errore
							Errore := ErrCOLLISIONE_PINZA;
							ErrCollisioneDebug := 27;			 
							RETURN; 
						END_IF	  
					END_IF 	
				{endregion}								   
				{Region "ROTAZIONE 90°" }
				ELSE	
					IF WorkAreaState^[iwa].Supporto.Tipologia = CAVALLETTO THEN 				
						IF (ModuleAX_Y^.Ax^.Status.ActPosition - IngombroDestinazioneY_Neg) <= (QuotaCentroPostazione + WorkAreaState^[iwa].Supporto.YDim/2) THEN //Se la pinza è in ingombro con il cavalletto nella zona a DX della sua metà
							QuotaFuoriIngombro_Y_Calcolata := MAX(QuotaFuoriIngombro_Y_Calcolata,
																QuotaCentroPostazione - 						(* Quota Y Postazione *)	
																// si Va con el eje a 0 grados no deve contemplar la pieza 16/7/2025																								
																//WorkAreaState^[iwa].Supporto.YDim/2 +	(* Dimensione/2 del Pallet/Cassa/Cavallina *)
																IngombroDestinazioneY_Neg 
																// si Va con el eje a 0 grados no deve contemplar la pieza 16/7/2025				   
																// + OffsetSicurezza.Y.Avuoto
																	);
						   NuIngombroYCalculado90G_Depuracion := 6 ;
							IF QuotaFuoriIngombro_Y_Calcolata + IngombroDestinazioneY_Pos >= WorkFootprint^[6].Y THEN//Se supero la quota massimo dell'area di lavoro genro un allarme
								Errore := ErrCOLLISIONE_PINZA;
								ErrCollisioneDebug := 28;			 
								RETURN; 
							END_IF 
						ELSIF (ModuleAX_Y^.Ax^.Status.ActPosition + IngombroDestinazioneY_Pos) >= (QuotaCentroPostazione - WorkAreaState^[iwa].Supporto.YDim/2) AND 
							(ModuleAX_Y^.Ax^.Status.ActPosition + IngombroDestinazioneY_Pos) <= (QuotaCentroPostazione) THEN //Se la pinza è in ingombro con il cavalletto con pinza dentro all'ingombro nella parte SX 
								QuotaFuoriIngombro_Y_Calcolata := MIN(QuotaFuoriIngombro_Y_Calcolata,
																	QuotaCentroPostazione - 						(* Quota Y Postazione *)																									
																	WorkAreaState^[iwa].Supporto.YDim/2 -	(* Dimensione/2 del Pallet/Cassa/Cavallina *)
																	IngombroDestinazioneY_Pos -
																	OffsetSicurezza.Y.Avuoto);
							   NuIngombroYCalculado90G_Depuracion := 7 ;
								IF QuotaFuoriIngombro_Y_Calcolata - IngombroDestinazioneY_Neg <= WorkArea^[iwa].Y + INGOMBRO_RISCONTRO_BUNDLE THEN//se sono dentro all'ingombro dei supporti del bundle genero un errore
									Errore := ErrCOLLISIONE_PINZA;
									ErrCollisioneDebug := 29;
									RETURN;										  
								END_IF 							
						ELSE
							QuotaFuoriIngombro_Y_Calcolata := MAX(QuotaFuoriIngombro_Y_Calcolata,
																QuotaCentroPostazione + 						(* Quota Y Postazione *)																									
																WorkAreaState^[iwa].Supporto.YDim/2 +	(* Dimensione/2 del Pallet/Cassa/Cavallina *)
																IngombroDestinazioneY_Neg +				(* Ingombro positivo pinza *)
																OffsetSicurezza.Y.Avuoto);				(* Offset sicurezza *)
						   NuIngombroYCalculado90G_Depuracion := 8 ;
							IF QuotaFuoriIngombro_Y_Calcolata - IngombroDestinazioneY_Neg <= WorkArea^[iwa].Y + INGOMBRO_RISCONTRO_BUNDLE THEN//se sono dentro all'ingombro dei supporti del bundle genero un errore
								Errore := ErrCOLLISIONE_PINZA;
								ErrCollisioneDebug := 30;
								RETURN;										  
							END_IF 
							IF QuotaFuoriIngombro_Y_Calcolata + IngombroDestinazioneY_Pos >= WorkFootprint^[6].Y THEN//Se supero la quota massimo dell'area di lavoro genro un allarme
								Errore := ErrCOLLISIONE_PINZA;
								ErrCollisioneDebug := 31;			 
								RETURN; 
							END_IF
						END_IF
					ELSIF WorkAreaState^[iwa].Supporto.Tipologia = BUNDLE THEN //se NELLA postazione c'è un bundle
						IF (ModuleAX_Y^.Ax^.Status.ActPosition - IngombroDestinazioneY_Neg) <= (QuotaCentroPostazione + INGOMBRO_RISCONTRO_BUNDLE) THEN //Se la pinza è dentro all'ingombro del bundle  
							QuotaFuoriIngombro_Y_Calcolata := MAX(QuotaFuoriIngombro_Y_Calcolata,
																	QuotaCentroPostazione + 					(* Quota Y Postazione *)																									
																	MAX(WorkAreaState^[iwa].Supporto.YDim,INGOMBRO_RISCONTRO_BUNDLE) + (* massimo tra Dimensione del bundle e dimensione riscontro *)
																	IngombroDestinazioneY_Neg +			(* Ingombro negativo pinza *)
																	OffsetSicurezza.Y.Avuoto);           (* Offset sicurezza *)
							NuIngombroYCalculado90G_Depuracion := 9 ;
							IF QuotaFuoriIngombro_Y_Calcolata - IngombroDestinazioneY_Neg <= WorkArea^[iwa].Y + INGOMBRO_RISCONTRO_BUNDLE THEN//se sono dentro all'ingombro dei supporti del bundle genero un errore
								Errore := ErrCOLLISIONE_PINZA;
								ErrCollisioneDebug := 32;
								RETURN;										  
							END_IF 
							IF QuotaFuoriIngombro_Y_Calcolata + IngombroDestinazioneY_Pos >= WorkFootprint^[6].Y THEN//Se supero la quota massimo dell'area di lavoro genro un allarme
								Errore := ErrCOLLISIONE_PINZA;
								ErrCollisioneDebug := 33;			 
								RETURN; 
							END_IF												  
						ELSE
							QuotaFuoriIngombro_Y_Calcolata := MAX(QuotaFuoriIngombro_Y_Calcolata,
																	QuotaCentroPostazione + 					(* Quota Y Postazione *)																									
																	MAX(WorkAreaState^[iwa].Supporto.YDim,INGOMBRO_RISCONTRO_BUNDLE) + (* massimo tra Dimensione del bundle e dimensione riscontro *)
																	//añadido 3_10_2025		
																	IngombroDestinazioneY_Pos  +			(* Ingombro negativo pinza *)
																	OffsetSicurezza.Y.Avuoto);           (* Offset sicurezza *)
						   NuIngombroYCalculado90G_Depuracion := 10 ;
							IF QuotaFuoriIngombro_Y_Calcolata - IngombroDestinazioneY_Neg <= QuotaCentroPostazione + INGOMBRO_RISCONTRO_BUNDLE THEN//se sono dentro all'ingombro dei supporti del bundle genero un errore
								Errore := ErrCOLLISIONE_PINZA;
								ErrCollisioneDebug := 34;
								RETURN;										  
							END_IF 
							IF QuotaFuoriIngombro_Y_Calcolata + IngombroDestinazioneY_Pos >= WorkFootprint^[6].Y THEN//Se supero la quota massimo dell'area di lavoro genro un allarme
								Errore := ErrCOLLISIONE_PINZA;
								ErrCollisioneDebug := 35;			 
								RETURN; 
							END_IF												  
						END_IF	
					ELSE//se non c'è nulla o c'è una cassa-pianale
						QuotaFuoriIngombro_Y_Calcolata := MAX(QuotaFuoriIngombro_Y_Calcolata,
										   						WorkArea^[iwa].Y + INGOMBRO_RISCONTRO_BUNDLE,//comunque devo sempre considerarlo perchè il riscontro è sempre presente!!!!
																MIN(ModuleAX_Y^.Ax^.Status.ActPosition,WorkFootprint^[6].Y - IngombroDestinazioneY_Pos - OffsetSicurezza.Y.Avuoto),
																WorkSpace^.Y/2 + OffSetPosYReposo+100);
					   NuIngombroYCalculado90G_Depuracion := 11 ;
						IF QuotaFuoriIngombro_Y_Calcolata + IngombroDestinazioneY_Pos >= WorkFootprint^[6].Y THEN//Se supero la quota massima dell'area di lavoro genro un allarme
							Errore := ErrCOLLISIONE_PINZA;
							ErrCollisioneDebug := 36;			 
							RETURN; 
						END_IF	
						IF QuotaFuoriIngombro_Y_Calcolata - IngombroDestinazioneY_Neg <= WorkArea^[iwa].Y + INGOMBRO_RISCONTRO_BUNDLE THEN//se sono dentro all'ingombro dei supporti del bundle genero un errore
							Errore := ErrCOLLISIONE_PINZA;
							ErrCollisioneDebug := 37;			 
							RETURN; 
						END_IF	  
					END_IF
				END_IF
				{endregion}				   
		{endregion}
		ELSE
			;//Errore.Code := ErrWAM_FTC_PostazioneNONDefinita;
		END_CASE
	{endregion}	
	ELSE
		;	
END_CASE
END_ACTION

ACTION CalcolaIngombroWALungoX:
/////////////////////////////////////////////////////////////!!!!!!!!!!!!!!!!!!!!!!!!!!!!!!!!//////////////////////////////
(*TFCalcolaNumeroPostazioneDXSX(PosizioneAttuale:=ModuleAX_X^.Ax^.Status.ActPosition,
								WorkArea:=WorkArea,
								DirezioneAsseX_Positiva:= TFDirezioneAssePositiva(Posizione_Attuale:=ModuleAX_X^.Ax^.Status.ActPosition,Posizione_Finale:=Mission^.XPick),
								NPostazioneDX=>WADX,
								NPostazioneSX=>WASX,
								PostazionePartenza=>WAPARTENZA);*)
								
AltezzaDiIngombroArea_CCENTRALE := 0;
AltezzaDiIngombroArea_CESTERNO := 0;
AltezzaDiIngombroArea_CESTERNO := 0;
FOR wa := 1 TO MAXAREAPRESENT DO
	
	CASE WorkArea^[wa].Typology OF
		TYPOLOGY_PALLET:
			CASE WorkAreaState^[wa].TransportState.Supporto.Tipologia OF
					
				PALLET_STANDARD:

					AltezzaDiIngombroArea_CCENTRALE := MAX(AltezzaDiIngombroArea_CCENTRALE, 
															WorkArea^[wa].Z +  MAX(//WorkArea^[wa].Z,
															WorkAreaState^[wa].H,
															WorkAreaState^[wa].HPL,
															WorkAreaState^[wa].TransportState.Supporto.HMAX,
															WorkAreaState^[wa].TransportState.Supporto.ZDim));

					AltezzaDiIngombroArea_CESTERNO	:= AltezzaDiIngombroArea_CCENTRALE;
					AltezzaDiIngombroArea_CINTERNO	:= AltezzaDiIngombroArea_CCENTRALE;
					
				PALLET_ACCOPPIATI:

					AltezzaDiIngombroArea_CCENTRALE := MAX(AltezzaDiIngombroArea_CCENTRALE, 
															WorkArea^[wa].Z +  MAX(//WorkArea^[wa].Z,
															WorkAreaState^[wa].H,
															WorkAreaState^[wa].HPL,
															WorkAreaState^[wa].TransportState.Supporto.HMAX,
															WorkAreaState^[wa].TransportState.Supporto.ZDim));

					AltezzaDiIngombroArea_CESTERNO	:= AltezzaDiIngombroArea_CCENTRALE;
					AltezzaDiIngombroArea_CINTERNO	:= AltezzaDiIngombroArea_CCENTRALE;
					
					
				CASSA_STANDARD:
									
					AltezzaDiIngombroArea_CCENTRALE := MAX(AltezzaDiIngombroArea_CCENTRALE, 
															WorkArea^[wa].Z +  MAX(//WorkArea^[wa].Z,
															WorkAreaState^[wa].H,
															WorkAreaState^[wa].HPL,
															WorkAreaState^[wa].TransportState.Supporto.HMAX,
															WorkAreaState^[wa].TransportState.Supporto.ZDim));

					AltezzaDiIngombroArea_CESTERNO	:= AltezzaDiIngombroArea_CCENTRALE;
					AltezzaDiIngombroArea_CINTERNO	:= AltezzaDiIngombroArea_CCENTRALE;
					
					
				CAVALLETTO:
					AltezzaDiIngombroArea_CCENTRALE := MAX(AltezzaDiIngombroArea_CCENTRALE, 
															WorkArea^[wa].Z,
															WorkAreaState^[wa].TransportState.Supporto.HMAX,
															WorkAreaState^[wa].TransportState.Supporto.ZDim);

					AltezzaDiIngombroArea_CESTERNO	:= MAX(AltezzaDiIngombroArea_CESTERNO,
															WorkArea^[wa].Z,
															//WorkAreaState^[wa].WorkPickPointTransportState.Supporto.HMAX,
															WorkAreaState^[wa].TransportState.Supporto.ZDim);

					AltezzaDiIngombroArea_CINTERNO	:= AltezzaDiIngombroArea_CESTERNO;
					
				BUNDLE:
					AltezzaDiIngombroArea_CCENTRALE := MAX(AltezzaDiIngombroArea_CCENTRALE, 
															WorkArea^[wa].Z,
															WorkAreaState^[wa].TransportState.Supporto.HMAX,
															WorkAreaState^[wa].TransportState.Supporto.ZDim);

					AltezzaDiIngombroArea_CESTERNO	:= MAX(AltezzaDiIngombroArea_CESTERNO,
															WorkArea^[wa].Z,
															//WorkAreaState^[wa].WorkPickPointTransportState.Supporto.HMAX,
															WorkAreaState^[wa].TransportState.Supporto.ZDim);

					AltezzaDiIngombroArea_CINTERNO	:= AltezzaDiIngombroArea_CESTERNO;
					
				ELSE
					AltezzaDiIngombroArea_CCENTRALE := WorkArea^[wa].Z;//Fisso l'altezza ad una quota di default
			END_CASE
						
		TYPOLOGY_LAYER:
			AltezzaDiIngombroArea_CCENTRALE := MAX(AltezzaDiIngombroArea_CCENTRALE,
													WorkArea^[wa].Z,
													WorkAreaState^[wa].H,
													WorkAreaState^[wa].HPL);

			AltezzaDiIngombroArea_CESTERNO	:= AltezzaDiIngombroArea_CCENTRALE;
			AltezzaDiIngombroArea_CINTERNO	:= AltezzaDiIngombroArea_CCENTRALE;
		
		TYPOLOGY_EXTERNAL_DEPPREL:
			AltezzaDiIngombroArea_CCENTRALE := AltezzaDiIngombroArea_CCENTRALE;
					
		TYPOLOGY_OVER_TRANSPORT:
			CASE WorkAreaState^[wa].TransportState.Supporto.Tipologia OF
					
				PALLET_STANDARD:

					AltezzaDiIngombroArea_CCENTRALE := MAX(AltezzaDiIngombroArea_CCENTRALE, 
															WorkArea^[wa].Z +  MAX(//WorkArea^[wa].Z,
															WorkAreaState^[wa].H,
															WorkAreaState^[wa].HPL,
															WorkAreaState^[wa].TransportState.Supporto.HMAX,
															WorkAreaState^[wa].TransportState.Supporto.ZDim));

					AltezzaDiIngombroArea_CESTERNO	:= AltezzaDiIngombroArea_CCENTRALE;
					AltezzaDiIngombroArea_CINTERNO	:= AltezzaDiIngombroArea_CCENTRALE;
					
				PALLET_ACCOPPIATI:

					AltezzaDiIngombroArea_CCENTRALE := MAX(AltezzaDiIngombroArea_CCENTRALE, 
															WorkArea^[wa].Z +  MAX(//WorkArea^[wa].Z,
															WorkAreaState^[wa].H,
															WorkAreaState^[wa].HPL,
															WorkAreaState^[wa].TransportState.Supporto.HMAX,
															WorkAreaState^[wa].TransportState.Supporto.ZDim));

					AltezzaDiIngombroArea_CESTERNO	:= AltezzaDiIngombroArea_CCENTRALE;
					AltezzaDiIngombroArea_CINTERNO	:= AltezzaDiIngombroArea_CCENTRALE;
	
				CASSA_STANDARD:
									
					AltezzaDiIngombroArea_CCENTRALE := MAX(AltezzaDiIngombroArea_CCENTRALE, 
															WorkArea^[wa].Z +  MAX(//WorkArea^[wa].Z,
															WorkAreaState^[wa].H,
															WorkAreaState^[wa].HPL,
															WorkAreaState^[wa].TransportState.Supporto.HMAX,
															WorkAreaState^[wa].TransportState.Supporto.ZDim));

					AltezzaDiIngombroArea_CESTERNO	:= AltezzaDiIngombroArea_CCENTRALE;
					AltezzaDiIngombroArea_CINTERNO	:= AltezzaDiIngombroArea_CCENTRALE;
					
					
				CAVALLETTO:
					AltezzaDiIngombroArea_CCENTRALE := MAX(AltezzaDiIngombroArea_CCENTRALE, 
															WorkArea^[wa].Z,
															WorkAreaState^[wa].TransportState.Supporto.HMAX,
															WorkAreaState^[wa].TransportState.Supporto.ZDim);

					AltezzaDiIngombroArea_CESTERNO	:= MAX(AltezzaDiIngombroArea_CESTERNO,
															WorkArea^[wa].Z,
															//WorkAreaState^[wa].WorkPickPointTransportState.Supporto.HMAX,
															WorkAreaState^[wa].TransportState.Supporto.ZDim);

					AltezzaDiIngombroArea_CINTERNO	:= AltezzaDiIngombroArea_CESTERNO;
					
				BUNDLE:
					AltezzaDiIngombroArea_CCENTRALE := MAX(AltezzaDiIngombroArea_CCENTRALE, 
															WorkArea^[wa].Z,
															WorkAreaState^[wa].TransportState.Supporto.HMAX,
															WorkAreaState^[wa].TransportState.Supporto.ZDim);

					AltezzaDiIngombroArea_CESTERNO	:= MAX(AltezzaDiIngombroArea_CESTERNO,
															WorkArea^[wa].Z,
															//WorkAreaState^[wa].WorkPickPointTransportState.Supporto.HMAX,
															WorkAreaState^[wa].TransportState.Supporto.ZDim);

					AltezzaDiIngombroArea_CINTERNO	:= AltezzaDiIngombroArea_CESTERNO;
				
				ELSE
					AltezzaDiIngombroArea_CCENTRALE := WorkArea^[wa].Z;//Fisso l'altezza ad una quota di default
			END_CASE
	END_CASE															
END_FOR	
		
(*ELSE
	(*TFCalcolaNumeroPostazioneDXSX(PosizioneAttuale	:= ModuleAX_X^.Ax^.Status.ActPosition,
									WorkArea		:= WorkArea,
									DirezioneAsseX_Positiva:=FALSE,
									NPostazioneDX	=> WADX,
									NPostazioneSX	=> WASX,
									PostazionePartenza=>WAPARTENZA);*)
			
	FOR wa := MAXAREA TO 1 BY -1 DO
		AltezzaDiIngombroArea_CCENTRALE := 0;
		IF WorkAreaState^[wa].H > WorkAreaState^[wa].HPL THEN
			AltezzaDiIngombroArea_CCENTRALE := WorkAreaState^[wa].H;
		ELSE
			AltezzaDiIngombroArea_CCENTRALE := WorkAreaState^[wa].HPL;
		END_IF
		IF QuotaFuoriIngombro_Z_AVUOTO_CCENTRALE <= AltezzaDiIngombroArea_CCENTRALE + TCPParameter.Z + OffsetSicurezza.Avuoto  THEN
			QuotaFuoriIngombro_Z_AVUOTO_CCENTRALE := AltezzaDiIngombroArea_CCENTRALE + TCPParameter.Z + OffsetSicurezza.Avuoto;
		END_IF
	END_FOR			
		(* Valuto I Pick-Point *)
		(*FOR P:=1 TO MAXPICKPOINT DO
			AltezzaDiIngombroPuntiPrelievo := 0;
			IF  WorkPickPoint^[P].Zh + WorkPickPointState^[P].ZDim >= WorkPickPointDimension[P].Zdim THEN // Se Altezza orrizzontale Ribaltino + Zpacco >= Ingombro Verticale Ribaltino
				AltezzaDiIngombroPuntiPrelievo := WorkPickPoint^[P].Zh + WorkPickPointState^[P].ZDim;
			END_IF
			IF WorkPickPoint^[P].Zv + WorkPickPointState^[P].ZTilter + WorkPickPointState^[P].YDim >= WorkPickPointDimension[P].Zdim THEN // Se Altezza Vertivale Ribaltino + Quota Fermo + Ypacco >= Ingombro Verticale Ribaltino
				AltezzaDiIngombroPuntiPrelievo := WorkPickPoint^[P].Zv + WorkPickPointState^[P].ZTilter + WorkPickPointState^[P].YDim;
			END_IF
			IF WorkPickPointDimension[P].Zdim >= AltezzaDiIngombroPuntiPrelievo THEN //Se Ingombro Verticale Ribaltino >= Dell'ingombro valutato sopra
				AltezzaDiIngombroPuntiPrelievo := WorkPickPointDimension[P].Zdim;
			END_IF
			IF WAPARTENZA = NPOSTAZIONE_PRIMADELPUNTODIPREL THEN //Se sono nella posizione 7 valuto l'altezza del ribaltino "REALE", con o senza pacco
				IF QuotaAnticipoDinamicaZ_VersoRiposo <= AltezzaDiIngombroPuntiPrelievo + TCPParameter.Z + OffsetSicurezza.Avuoto THEN //Se Quota fuori ingombro <= dell' ingombro del punto di prelievo
					QuotaAnticipoDinamicaZ_VersoRiposo := AltezzaDiIngombroPuntiPrelievo + TCPParameter.Z + OffsetSicurezza.Avuoto;
				END_IF
			ELSE		//Se non sono nella WA 7, do una quota fittizzia, inferiore all'altezza del ribaltino "reale"
				IF QuotaAnticipoDinamicaZ_VersoRiposo <= AltezzaDiIngombroPuntiPrelievo + TCPParameter.Z + OffsetSicurezzaAnticipoMovimenti.OffsetSicurezzaAnticipo_Z - 300 THEN
					QuotaAnticipoDinamicaZ_VersoRiposo := AltezzaDiIngombroPuntiPrelievo + WorkPickPointState^[P].YDim + TCPParameter.Z + OffsetSicurezzaAnticipoMovimenti.OffsetSicurezzaAnticipo_Z - 300;
				END_IF
			END_IF
		END_FOR*)
	//END_IF
	IF ModuleAX_Z^.Ax^.Status.ActPosition >= QuotaAnticipoDinamicaZ_VersoRiposo THEN
		QuotaAnticipoDinamicaZ_Raggiunta := TRUE;
	ELSE
		QuotaAnticipoDinamicaZ_Raggiunta := FALSE;
	END_IF



END_IF*)
END_ACTION

ACTION CalcolaIngombroWALungoX_Pal:
								
AltezzaDiIngombroArea_CCENTRALE := 0;
AltezzaDiIngombroArea_CESTERNO := 0;
AltezzaDiIngombroArea_CESTERNO := 0;
FOR wa := 1 TO MAXAREAPRESENT DO
	
	CASE WorkArea^[wa].Typology OF
		TYPOLOGY_PALLET:
			CASE WorkAreaState^[wa].Supporto.Tipologia OF
					
				PALLET_STANDARD:

					AltezzaDiIngombroArea_CCENTRALE := MAX(AltezzaDiIngombroArea_CCENTRALE, 
															WorkArea^[wa].Z +  MAX(//WorkArea^[wa].Z,
															WorkAreaState^[wa].H,
															WorkAreaState^[wa].HPL,
															WorkAreaState^[wa].Supporto.HMAX,
															WorkAreaState^[wa].Supporto.ZDim));

					AltezzaDiIngombroArea_CESTERNO	:= AltezzaDiIngombroArea_CCENTRALE;
					AltezzaDiIngombroArea_CINTERNO	:= AltezzaDiIngombroArea_CCENTRALE;
					
				PALLET_ACCOPPIATI:

					AltezzaDiIngombroArea_CCENTRALE := MAX(AltezzaDiIngombroArea_CCENTRALE, 
															WorkArea^[wa].Z +  MAX(//WorkArea^[wa].Z,
															WorkAreaState^[wa].H,
															WorkAreaState^[wa].HPL,
															WorkAreaState^[wa].Supporto.HMAX,
															WorkAreaState^[wa].Supporto.ZDim));

					AltezzaDiIngombroArea_CESTERNO	:= AltezzaDiIngombroArea_CCENTRALE;
					AltezzaDiIngombroArea_CINTERNO	:= AltezzaDiIngombroArea_CCENTRALE;
					
					
				CASSA_STANDARD:
									
					AltezzaDiIngombroArea_CCENTRALE := MAX(AltezzaDiIngombroArea_CCENTRALE, 
															WorkArea^[wa].Z +  MAX(//WorkArea^[wa].Z,
															WorkAreaState^[wa].H,
															WorkAreaState^[wa].HPL,
															WorkAreaState^[wa].Supporto.HMAX,
															WorkAreaState^[wa].Supporto.ZDim));

					AltezzaDiIngombroArea_CESTERNO	:= AltezzaDiIngombroArea_CCENTRALE;
					AltezzaDiIngombroArea_CINTERNO	:= AltezzaDiIngombroArea_CCENTRALE;
					
					
				CAVALLETTO:
					AltezzaDiIngombroArea_CCENTRALE := MAX(AltezzaDiIngombroArea_CCENTRALE, 
															WorkArea^[wa].Z,
															//WorkAreaState^[wa].Supporto.HMAX,
															WorkAreaState^[wa].Supporto.ZDim);

					AltezzaDiIngombroArea_CESTERNO	:= MAX(AltezzaDiIngombroArea_CESTERNO,
															WorkArea^[wa].Z,
															//WorkAreaState^[wa].WorkPickPointTransportState.Supporto.HMAX,
															WorkAreaState^[wa].Supporto.ZDim);

					AltezzaDiIngombroArea_CINTERNO	:= AltezzaDiIngombroArea_CESTERNO;
					
				BUNDLE:
					AltezzaDiIngombroArea_CCENTRALE := MAX(AltezzaDiIngombroArea_CCENTRALE, 
															WorkArea^[wa].Z,
															//WorkAreaState^[wa].Supporto.HMAX,
															WorkAreaState^[wa].Supporto.ZDim);

					AltezzaDiIngombroArea_CESTERNO	:= MAX(AltezzaDiIngombroArea_CESTERNO,
															WorkArea^[wa].Z,
															//WorkAreaState^[wa].WorkPickPointTransportState.Supporto.HMAX,
															WorkAreaState^[wa].Supporto.ZDim);

					AltezzaDiIngombroArea_CINTERNO	:= AltezzaDiIngombroArea_CESTERNO;
					
				ELSE
					AltezzaDiIngombroArea_CCENTRALE := WorkArea^[wa].Z;//Fisso l'altezza ad una quota di default
			END_CASE
						
		TYPOLOGY_LAYER:
			AltezzaDiIngombroArea_CCENTRALE := MAX(AltezzaDiIngombroArea_CCENTRALE,
													WorkArea^[wa].Z,
													WorkAreaState^[wa].H,
													WorkAreaState^[wa].HPL);

			AltezzaDiIngombroArea_CESTERNO	:= AltezzaDiIngombroArea_CCENTRALE;
			AltezzaDiIngombroArea_CINTERNO	:= AltezzaDiIngombroArea_CCENTRALE;
		
		TYPOLOGY_EXTERNAL_DEPPREL:
			AltezzaDiIngombroArea_CCENTRALE := AltezzaDiIngombroArea_CCENTRALE;
					
		TYPOLOGY_OVER_TRANSPORT:
			CASE WorkAreaState^[wa].Supporto.Tipologia OF
					
				PALLET_STANDARD:

					AltezzaDiIngombroArea_CCENTRALE := MAX(AltezzaDiIngombroArea_CCENTRALE, 
															WorkArea^[wa].Z +  MAX(//WorkArea^[wa].Z,
															WorkAreaState^[wa].H,
															WorkAreaState^[wa].HPL,
															WorkAreaState^[wa].Supporto.HMAX,
															WorkAreaState^[wa].Supporto.ZDim));

					AltezzaDiIngombroArea_CESTERNO	:= AltezzaDiIngombroArea_CCENTRALE;
					AltezzaDiIngombroArea_CINTERNO	:= AltezzaDiIngombroArea_CCENTRALE;
					
				PALLET_ACCOPPIATI:

					AltezzaDiIngombroArea_CCENTRALE := MAX(AltezzaDiIngombroArea_CCENTRALE, 
															WorkArea^[wa].Z +  MAX(//WorkArea^[wa].Z,
															WorkAreaState^[wa].H,
															WorkAreaState^[wa].HPL,
															WorkAreaState^[wa].Supporto.HMAX,
															WorkAreaState^[wa].Supporto.ZDim));

					AltezzaDiIngombroArea_CESTERNO	:= AltezzaDiIngombroArea_CCENTRALE;
					AltezzaDiIngombroArea_CINTERNO	:= AltezzaDiIngombroArea_CCENTRALE;
	
				CASSA_STANDARD:
									
					AltezzaDiIngombroArea_CCENTRALE := MAX(AltezzaDiIngombroArea_CCENTRALE, 
															WorkArea^[wa].Z +  MAX(//WorkArea^[wa].Z,
															WorkAreaState^[wa].H,
															WorkAreaState^[wa].HPL,
															WorkAreaState^[wa].Supporto.HMAX,
															WorkAreaState^[wa].Supporto.ZDim));

					AltezzaDiIngombroArea_CESTERNO	:= AltezzaDiIngombroArea_CCENTRALE;
					AltezzaDiIngombroArea_CINTERNO	:= AltezzaDiIngombroArea_CCENTRALE;
					
					
				CAVALLETTO:
					AltezzaDiIngombroArea_CCENTRALE := MAX(AltezzaDiIngombroArea_CCENTRALE, 
															WorkArea^[wa].Z,
															WorkAreaState^[wa].Supporto.HMAX,
															WorkAreaState^[wa].Supporto.ZDim);

					AltezzaDiIngombroArea_CESTERNO	:= MAX(AltezzaDiIngombroArea_CESTERNO,
															WorkArea^[wa].Z,
															//WorkAreaState^[wa].WorkPickPointTransportState.Supporto.HMAX,
															WorkAreaState^[wa].Supporto.ZDim);

					AltezzaDiIngombroArea_CINTERNO	:= AltezzaDiIngombroArea_CESTERNO;
					
				BUNDLE:
					AltezzaDiIngombroArea_CCENTRALE := MAX(AltezzaDiIngombroArea_CCENTRALE, 
															WorkArea^[wa].Z,
															WorkAreaState^[wa].Supporto.HMAX,
															WorkAreaState^[wa].Supporto.ZDim);

					AltezzaDiIngombroArea_CESTERNO	:= MAX(AltezzaDiIngombroArea_CESTERNO,
															WorkArea^[wa].Z,
															//WorkAreaState^[wa].WorkPickPointTransportState.Supporto.HMAX,
															WorkAreaState^[wa].Supporto.ZDim);

					AltezzaDiIngombroArea_CINTERNO	:= AltezzaDiIngombroArea_CESTERNO;
				
				ELSE
					AltezzaDiIngombroArea_CCENTRALE := WorkArea^[wa].Z;//Fisso l'altezza ad una quota di default
			END_CASE
	END_CASE															
END_FOR
END_ACTION

ACTION CalcolaIngombroWALungoY:
AltezzaDiIngombroArea_CCENTRALE := 0;
AltezzaDiIngombroArea_CESTERNO := 0;
AltezzaDiIngombroArea_CESTERNO := 0;
FOR wa := 1 TO MAXAREAPRESENT DO
	IF AbilitaValutazioneFISuSingolaWA AND NumeroWAValutazioneFISingolaPostazione > 0 THEN
		wa := NumeroWAValutazioneFISingolaPostazione; 	
	END_IF
	CASE WorkArea^[wa].Typology OF
		TYPOLOGY_PALLET:
			CASE WorkAreaState^[wa].TransportState.Supporto.Tipologia OF
					
				PALLET_STANDARD:

					AltezzaDiIngombroArea_CCENTRALE := MAX(AltezzaDiIngombroArea_CCENTRALE, 
															WorkArea^[wa].Z +  MAX(//WorkArea^[wa].Z,
															WorkAreaState^[wa].H,
															WorkAreaState^[wa].HPL,
															WorkAreaState^[wa].TransportState.Supporto.HMAX,
															WorkAreaState^[wa].TransportState.Supporto.ZDim));

					AltezzaDiIngombroArea_CESTERNO	:= AltezzaDiIngombroArea_CCENTRALE;
					AltezzaDiIngombroArea_CINTERNO	:= AltezzaDiIngombroArea_CCENTRALE;
				
				PALLET_ACCOPPIATI:

					AltezzaDiIngombroArea_CCENTRALE := MAX(AltezzaDiIngombroArea_CCENTRALE, 
															WorkArea^[wa].Z +  MAX(//WorkArea^[wa].Z,
															WorkAreaState^[wa].H,
															WorkAreaState^[wa].HPL,
															WorkAreaState^[wa].TransportState.Supporto.HMAX,
															WorkAreaState^[wa].TransportState.Supporto.ZDim));

					AltezzaDiIngombroArea_CESTERNO	:= AltezzaDiIngombroArea_CCENTRALE;
					AltezzaDiIngombroArea_CINTERNO	:= AltezzaDiIngombroArea_CCENTRALE;				
	
				CASSA_STANDARD:
									
					AltezzaDiIngombroArea_CCENTRALE := MAX(AltezzaDiIngombroArea_CCENTRALE, 
															WorkArea^[wa].Z +  MAX(//WorkArea^[wa].Z,
															WorkAreaState^[wa].H,
															WorkAreaState^[wa].HPL,
															WorkAreaState^[wa].TransportState.Supporto.HMAX,
															WorkAreaState^[wa].TransportState.Supporto.ZDim));

					AltezzaDiIngombroArea_CESTERNO	:= AltezzaDiIngombroArea_CCENTRALE;
					AltezzaDiIngombroArea_CINTERNO	:= AltezzaDiIngombroArea_CCENTRALE;
					
					
				CAVALLETTO:
					AltezzaDiIngombroArea_CCENTRALE := MAX(AltezzaDiIngombroArea_CCENTRALE, 
															WorkArea^[wa].Z,
															//WorkAreaState^[wa].WorkPickPointTransportState.Supporto.HMAX,
															WorkAreaState^[wa].TransportState.Supporto.ZDim);

					AltezzaDiIngombroArea_CESTERNO	:= MAX(AltezzaDiIngombroArea_CESTERNO,
															WorkArea^[wa].Z,
															//WorkAreaState^[wa].WorkPickPointTransportState.Supporto.HMAX,
															WorkAreaState^[wa].TransportState.Supporto.ZDim);

					AltezzaDiIngombroArea_CINTERNO	:= AltezzaDiIngombroArea_CESTERNO;
					
				BUNDLE:
					AltezzaDiIngombroArea_CCENTRALE := MAX(AltezzaDiIngombroArea_CCENTRALE, 
															WorkArea^[wa].Z,
															//WorkAreaState^[wa].WorkPickPointTransportState.Supporto.HMAX,
															WorkAreaState^[wa].TransportState.Supporto.ZDim);

					AltezzaDiIngombroArea_CESTERNO	:= MAX(AltezzaDiIngombroArea_CESTERNO,
															WorkArea^[wa].Z,
															//WorkAreaState^[wa].WorkPickPointTransportState.Supporto.HMAX,
															WorkAreaState^[wa].TransportState.Supporto.ZDim);

					AltezzaDiIngombroArea_CINTERNO	:= AltezzaDiIngombroArea_CESTERNO;	
					
				ELSE
					AltezzaDiIngombroArea_CCENTRALE := WorkArea^[wa].Z;;//Fisso l'altezza ad una quota di default
			END_CASE
						
		TYPOLOGY_LAYER:
			AltezzaDiIngombroArea_CCENTRALE := MAX(AltezzaDiIngombroArea_CCENTRALE,
													WorkArea^[wa].Z,
													WorkAreaState^[wa].H,
													WorkAreaState^[wa].HPL);

			AltezzaDiIngombroArea_CESTERNO	:= AltezzaDiIngombroArea_CCENTRALE;
			AltezzaDiIngombroArea_CINTERNO	:= AltezzaDiIngombroArea_CCENTRALE;
		
		TYPOLOGY_EXTERNAL_DEPPREL:
			AltezzaDiIngombroArea_CCENTRALE := AltezzaDiIngombroArea_CCENTRALE;
					
		TYPOLOGY_OVER_TRANSPORT:
			CASE WorkAreaState^[wa].TransportState.Supporto.Tipologia OF
					
				PALLET_STANDARD:

					AltezzaDiIngombroArea_CCENTRALE := MAX(AltezzaDiIngombroArea_CCENTRALE, 
															WorkArea^[wa].Z +  MAX(//WorkArea^[wa].Z,
															WorkAreaState^[wa].H,
															WorkAreaState^[wa].HPL,
															WorkAreaState^[wa].TransportState.Supporto.HMAX,
															WorkAreaState^[wa].TransportState.Supporto.ZDim));

					AltezzaDiIngombroArea_CESTERNO	:= AltezzaDiIngombroArea_CCENTRALE;
					AltezzaDiIngombroArea_CINTERNO	:= AltezzaDiIngombroArea_CCENTRALE;
					
				PALLET_ACCOPPIATI:

					AltezzaDiIngombroArea_CCENTRALE := MAX(AltezzaDiIngombroArea_CCENTRALE, 
															WorkArea^[wa].Z +  MAX(//WorkArea^[wa].Z,
															WorkAreaState^[wa].H,
															WorkAreaState^[wa].HPL,
															WorkAreaState^[wa].TransportState.Supporto.HMAX,
															WorkAreaState^[wa].TransportState.Supporto.ZDim));

					AltezzaDiIngombroArea_CESTERNO	:= AltezzaDiIngombroArea_CCENTRALE;
					AltezzaDiIngombroArea_CINTERNO	:= AltezzaDiIngombroArea_CCENTRALE;	
					
				CASSA_STANDARD:
									
					AltezzaDiIngombroArea_CCENTRALE := MAX(AltezzaDiIngombroArea_CCENTRALE, 
															WorkArea^[wa].Z +  MAX(//WorkArea^[wa].Z,
															WorkAreaState^[wa].H,
															WorkAreaState^[wa].HPL,
															WorkAreaState^[wa].TransportState.Supporto.HMAX,
															WorkAreaState^[wa].TransportState.Supporto.ZDim));

					AltezzaDiIngombroArea_CESTERNO	:= AltezzaDiIngombroArea_CCENTRALE;
					AltezzaDiIngombroArea_CINTERNO	:= AltezzaDiIngombroArea_CCENTRALE;
					
					
				CAVALLETTO:
					AltezzaDiIngombroArea_CCENTRALE := MAX(AltezzaDiIngombroArea_CCENTRALE, 
															WorkArea^[wa].Z,
															//WorkAreaState^[wa].WorkPickPointTransportState.Supporto.HMAX,
															WorkAreaState^[wa].TransportState.Supporto.ZDim);

					AltezzaDiIngombroArea_CESTERNO	:= MAX(AltezzaDiIngombroArea_CESTERNO,
															WorkArea^[wa].Z,
															//WorkAreaState^[wa].WorkPickPointTransportState.Supporto.HMAX,
															WorkAreaState^[wa].TransportState.Supporto.ZDim);

					AltezzaDiIngombroArea_CINTERNO	:= AltezzaDiIngombroArea_CESTERNO;
					
				BUNDLE:
					AltezzaDiIngombroArea_CCENTRALE := MAX(AltezzaDiIngombroArea_CCENTRALE, 
															WorkArea^[wa].Z,
															//WorkAreaState^[wa].WorkPickPointTransportState.Supporto.HMAX,
															WorkAreaState^[wa].TransportState.Supporto.ZDim);

					AltezzaDiIngombroArea_CESTERNO	:= MAX(AltezzaDiIngombroArea_CESTERNO,
															WorkArea^[wa].Z,
															//WorkAreaState^[wa].WorkPickPointTransportState.Supporto.HMAX,
															WorkAreaState^[wa].TransportState.Supporto.ZDim);

					AltezzaDiIngombroArea_CINTERNO	:= AltezzaDiIngombroArea_CESTERNO;
				
				ELSE
					AltezzaDiIngombroArea_CCENTRALE := WorkArea^[wa].Z;;//Fisso l'altezza ad una quota di default
			END_CASE
	END_CASE	
	IF 	AbilitaValutazioneFISuSingolaWA AND NumeroWAValutazioneFISingolaPostazione > 0 THEN
		RETURN; 	
	END_IF														
END_FOR
END_ACTION

ACTION CalcolaIngombroWALungoY_Pal:
AltezzaDiIngombroArea_CCENTRALE := 0;
AltezzaDiIngombroArea_CESTERNO := 0;
AltezzaDiIngombroArea_CESTERNO := 0;
FOR wa := 1 TO MAXAREAPRESENT DO
	IF AbilitaValutazioneFISuSingolaWA AND NumeroWAValutazioneFISingolaPostazione > 0 THEN
		wa := NumeroWAValutazioneFISingolaPostazione; 	
	END_IF
	CASE WorkArea^[wa].Typology OF
		TYPOLOGY_PALLET:
			CASE WorkAreaState^[wa].TransportState.Supporto.Tipologia OF
					
				PALLET_STANDARD:

					AltezzaDiIngombroArea_CCENTRALE := MAX(AltezzaDiIngombroArea_CCENTRALE, 
															WorkArea^[wa].Z +  MAX(//WorkArea^[wa].Z,
															WorkAreaState^[wa].H,
															WorkAreaState^[wa].HPL,
															WorkAreaState^[wa].TransportState.Supporto.HMAX,
															WorkAreaState^[wa].TransportState.Supporto.ZDim));

					AltezzaDiIngombroArea_CESTERNO	:= AltezzaDiIngombroArea_CCENTRALE;
					AltezzaDiIngombroArea_CINTERNO	:= AltezzaDiIngombroArea_CCENTRALE;
				
				PALLET_ACCOPPIATI:

					AltezzaDiIngombroArea_CCENTRALE := MAX(AltezzaDiIngombroArea_CCENTRALE, 
															WorkArea^[wa].Z +  MAX(//WorkArea^[wa].Z,
															WorkAreaState^[wa].H,
															WorkAreaState^[wa].HPL,
															WorkAreaState^[wa].TransportState.Supporto.HMAX,
															WorkAreaState^[wa].TransportState.Supporto.ZDim));

					AltezzaDiIngombroArea_CESTERNO	:= AltezzaDiIngombroArea_CCENTRALE;
					AltezzaDiIngombroArea_CINTERNO	:= AltezzaDiIngombroArea_CCENTRALE;				
	
				CASSA_STANDARD:
									
					AltezzaDiIngombroArea_CCENTRALE := MAX(AltezzaDiIngombroArea_CCENTRALE, 
															WorkArea^[wa].Z +  MAX(//WorkArea^[wa].Z,
															WorkAreaState^[wa].H,
															WorkAreaState^[wa].HPL,
															WorkAreaState^[wa].TransportState.Supporto.HMAX,
															WorkAreaState^[wa].TransportState.Supporto.ZDim));

					AltezzaDiIngombroArea_CESTERNO	:= AltezzaDiIngombroArea_CCENTRALE;
					AltezzaDiIngombroArea_CINTERNO	:= AltezzaDiIngombroArea_CCENTRALE;
					
					
				CAVALLETTO:
					AltezzaDiIngombroArea_CCENTRALE := MAX(AltezzaDiIngombroArea_CCENTRALE, 
															WorkArea^[wa].Z,
															//WorkAreaState^[wa].WorkPickPointTransportState.Supporto.HMAX,
															WorkAreaState^[wa].TransportState.Supporto.ZDim);

					AltezzaDiIngombroArea_CESTERNO	:= MAX(AltezzaDiIngombroArea_CESTERNO,
															WorkArea^[wa].Z,
															//WorkAreaState^[wa].WorkPickPointTransportState.Supporto.HMAX,
															WorkAreaState^[wa].TransportState.Supporto.ZDim);

					AltezzaDiIngombroArea_CINTERNO	:= AltezzaDiIngombroArea_CESTERNO;
					
				BUNDLE:
					AltezzaDiIngombroArea_CCENTRALE := MAX(AltezzaDiIngombroArea_CCENTRALE, 
															WorkArea^[wa].Z,
															//WorkAreaState^[wa].WorkPickPointTransportState.Supporto.HMAX,
															WorkAreaState^[wa].TransportState.Supporto.ZDim);

					AltezzaDiIngombroArea_CESTERNO	:= MAX(AltezzaDiIngombroArea_CESTERNO,
															WorkArea^[wa].Z,
															//WorkAreaState^[wa].WorkPickPointTransportState.Supporto.HMAX,
															WorkAreaState^[wa].TransportState.Supporto.ZDim);

					AltezzaDiIngombroArea_CINTERNO	:= AltezzaDiIngombroArea_CESTERNO;
					
				ELSE
					AltezzaDiIngombroArea_CCENTRALE := WorkArea^[wa].Z;;//Fisso l'altezza ad una quota di default
			END_CASE
						
		TYPOLOGY_LAYER:
			AltezzaDiIngombroArea_CCENTRALE := MAX(AltezzaDiIngombroArea_CCENTRALE,
													WorkArea^[wa].Z,
													WorkAreaState^[wa].H,
													WorkAreaState^[wa].HPL);

			AltezzaDiIngombroArea_CESTERNO	:= AltezzaDiIngombroArea_CCENTRALE;
			AltezzaDiIngombroArea_CINTERNO	:= AltezzaDiIngombroArea_CCENTRALE;
		
		TYPOLOGY_EXTERNAL_DEPPREL:
			AltezzaDiIngombroArea_CCENTRALE := AltezzaDiIngombroArea_CCENTRALE;
					
		TYPOLOGY_OVER_TRANSPORT:
			CASE WorkAreaState^[wa].TransportState.Supporto.Tipologia OF
					
				PALLET_STANDARD:

					AltezzaDiIngombroArea_CCENTRALE := MAX(AltezzaDiIngombroArea_CCENTRALE, 
															WorkArea^[wa].Z +  MAX(//WorkArea^[wa].Z,
															WorkAreaState^[wa].H,
															WorkAreaState^[wa].HPL,
															WorkAreaState^[wa].TransportState.Supporto.HMAX,
															WorkAreaState^[wa].TransportState.Supporto.ZDim));

					AltezzaDiIngombroArea_CESTERNO	:= AltezzaDiIngombroArea_CCENTRALE;
					AltezzaDiIngombroArea_CINTERNO	:= AltezzaDiIngombroArea_CCENTRALE;
					
				PALLET_ACCOPPIATI:

					AltezzaDiIngombroArea_CCENTRALE := MAX(AltezzaDiIngombroArea_CCENTRALE, 
															WorkArea^[wa].Z +  MAX(//WorkArea^[wa].Z,
															WorkAreaState^[wa].H,
															WorkAreaState^[wa].HPL,
															WorkAreaState^[wa].TransportState.Supporto.HMAX,
															WorkAreaState^[wa].TransportState.Supporto.ZDim));

					AltezzaDiIngombroArea_CESTERNO	:= AltezzaDiIngombroArea_CCENTRALE;
					AltezzaDiIngombroArea_CINTERNO	:= AltezzaDiIngombroArea_CCENTRALE;	
					
				CASSA_STANDARD:
									
					AltezzaDiIngombroArea_CCENTRALE := MAX(AltezzaDiIngombroArea_CCENTRALE, 
															WorkArea^[wa].Z +  MAX(//WorkArea^[wa].Z,
															WorkAreaState^[wa].H,
															WorkAreaState^[wa].HPL,
															WorkAreaState^[wa].TransportState.Supporto.HMAX,
															WorkAreaState^[wa].TransportState.Supporto.ZDim));

					AltezzaDiIngombroArea_CESTERNO	:= AltezzaDiIngombroArea_CCENTRALE;
					AltezzaDiIngombroArea_CINTERNO	:= AltezzaDiIngombroArea_CCENTRALE;
					
					
				CAVALLETTO:
					AltezzaDiIngombroArea_CCENTRALE := MAX(AltezzaDiIngombroArea_CCENTRALE, 
															WorkArea^[wa].Z,
															//WorkAreaState^[wa].WorkPickPointTransportState.Supporto.HMAX,
															WorkAreaState^[wa].TransportState.Supporto.ZDim);

					AltezzaDiIngombroArea_CESTERNO	:= MAX(AltezzaDiIngombroArea_CESTERNO,
															WorkArea^[wa].Z,
															//WorkAreaState^[wa].WorkPickPointTransportState.Supporto.HMAX,
															WorkAreaState^[wa].TransportState.Supporto.ZDim);

					AltezzaDiIngombroArea_CINTERNO	:= AltezzaDiIngombroArea_CESTERNO;
				
				BUNDLE:
					AltezzaDiIngombroArea_CCENTRALE := MAX(AltezzaDiIngombroArea_CCENTRALE, 
															WorkArea^[wa].Z,
															//WorkAreaState^[wa].WorkPickPointTransportState.Supporto.HMAX,
															WorkAreaState^[wa].TransportState.Supporto.ZDim);

					AltezzaDiIngombroArea_CESTERNO	:= MAX(AltezzaDiIngombroArea_CESTERNO,
															WorkArea^[wa].Z,
															//WorkAreaState^[wa].WorkPickPointTransportState.Supporto.HMAX,
															WorkAreaState^[wa].TransportState.Supporto.ZDim);

					AltezzaDiIngombroArea_CINTERNO	:= AltezzaDiIngombroArea_CESTERNO;
				
				ELSE
					AltezzaDiIngombroArea_CCENTRALE := WorkArea^[wa].Z;;//Fisso l'altezza ad una quota di default
			END_CASE
	END_CASE	
	IF 	AbilitaValutazioneFISuSingolaWA AND NumeroWAValutazioneFISingolaPostazione > 0 THEN
		RETURN; 	
	END_IF														
END_FOR
END_ACTION

ACTION CalcoloFuriIngombroVerticale:
(* Calcolo gli ingombri della pinza nelle varie direzioni *)
TFCalcoliIngombroPinza(Mission := Mission,
					WorkAreaManager := WorkAreaManager,
					WorkAreaState := ADR(WorkAreaState),
					ModuleAX_J := ModuleAX_J,
					AngoloRotazioneDestinazionePinza:= AngoloRotazioneDestinazionePinza,
					IngombroX_Pos := ADR(IngombroX_Pos),
					IngombroY_Pos := ADR(IngombroY_Pos),
					IngombroX_Neg := ADR(IngombroX_Neg),
					IngombroY_Neg := ADR(IngombroY_Neg),
					IngombroZ_Pos := ADR(IngombroZ_Pos),
					IngombroZ_Neg := ADR(IngombroZ_Neg),
					IngombroY_Tot := ADR(IngombroY_Tot),
					IngombroDestinazioneX_Pos := ADR(IngombroDestinazioneX_Pos),
					IngombroDestinazioneY_Pos := ADR(IngombroDestinazioneY_Pos),
					IngombroDestinazioneX_Neg := ADR(IngombroDestinazioneX_Neg),
					IngombroDestinazioneY_Neg := ADR(IngombroDestinazioneY_Neg),
					IngombroDestinazioneZ_Pos := ADR(IngombroDestinazioneZ_Pos),
					IngombroDestinazioneZ_Neg := ADR(IngombroDestinazioneZ_Neg),
					IngombroMaxX_Pos := ADR(IngombroMaxX_Pos),
					IngombroMaxY_Pos := ADR(IngombroMaxY_Pos),
					IngombroMaxX_Neg := ADR(IngombroMaxX_Neg),
					IngombroMaxY_Neg := ADR(IngombroMaxY_Neg),
					IngombroMaxZ_Pos := ADR(IngombroMaxZ_Pos),
					IngombroMaxZ_Neg := ADR(IngombroMaxZ_Neg),
					IngombroY_Pos_0  	:= ADR(IngombroY_Pos_0),		 		
					IngombroY_Neg_180 	:= ADR(IngombroY_Neg_180),
					IngombroY_Neg_0 	:= ADR(IngombroY_Neg_0),	
					IngombroY_Pos_180 	:= ADR(IngombroY_Pos_180),
					ScostamentoVerticalePuntoCentrale := ADR(ScostamentoVerticalePuntoCentrale));


	
////////////FI Asse Z
QuotaFuoriIngombro_Z_AVUOTO_CCENTRALE 	:= 0;
QuotaFuoriIngombro_Z_AVUOTO_CESTERNO 	:= 0;
QuotaFuoriIngombro_Z_AVUOTO_CINTERNO 	:= 0;
AltezzaDiIngombroPuntiPrelievo := 0;
AltezzaDiIngombroIngombri_CCENTRALE := 0;
(* Valuto gli ostacoli *)	
FOR f:=1 TO MAXFOOTPRINT DO
	AltezzaDiIngombroIngombri_CCENTRALE := MAX(AltezzaDiIngombroIngombri_CCENTRALE,WorkFootPrint^[f].Z + WorkFootPrint^[f].ZDim);// + IngombroMaxZ_Neg);
END_FOR

(* Valuto I Pick-Point *)
FOR P:=1 TO MAXPICKPOINT DO	
	AltezzaDiIngombroPuntiPrelievo := MAX(AltezzaDiIngombroPuntiPrelievo,WorkPickPointDimension^[P].Zdim,WorkPickPoint^[P].ZRaise,WorkPickPoint^[P].Z);
END_FOR

(* Valuto le wa *)			
CASE ASSE_DISPOSIZIONE_POSTAZIONI OF
	
	LUNGO_X:
			CalcolaIngombroWALungoX_Pal();
	
	LUNGO_Y:
			CalcolaIngombroWALungoY_Pal();

END_CASE

(*
(* Valuto se gli assi sono in finestra di prelievo, in questo modo valuto nel ciclo se devo andare fuori ingombro oppure posso partire da dove sono *)
AsseXInFinestraDiPrelievo := FALSE;
IF (ModuleAx_X^.Ax^.AxRef^.NcToPlc.ActPos >= Mission^.XPick - 50) AND (ModuleAx_X^.Ax^.AxRef^.NcToPlc.ActPos <=  Mission^.XPick + 50) THEN
	AsseXInFinestraDiPrelievo := TRUE;
END_IF
AsseYInFinestraDiPrelievo := FALSE;
IF (ModuleAx_Y^.Ax^.AxRef^.NcToPlc.ActPos  >=  Mission^.YPick - 50) AND (ModuleAx_Y^.Ax^.AxRef^.NcToPlc.SetPos <= Mission^.YPick + 50) THEN
	AsseYInFinestraDiPrelievo := TRUE;
END_IF
(* Valuto la rotazione della pinza *)
AsseJInFinestraDiPrelievo := FALSE;
IF ModuleAx_J^.Ax^.AxRef^.NcToPlc.ActPos >= Mission^.JPick - 5 AND ModuleAx_J^.Ax^.AxRef^.NcToPlc.ActPos <= Mission^.JPick + 5 THEN
	AsseJInFinestraDiPrelievo := TRUE;
END_IF*)
END_ACTION

END_FUNCTION_BLOCK

// ---- POUs/TFPalletizerDataTF/Utility Varie/TFCalcolaQuotaIngombroColonneLastre.TcPOU
FUNCTION_BLOCK TFCalcolaQuotaIngombroColonneLastre
VAR_INPUT
	QuotaY_ColonnaDX : LREAL; 		(* Quota della colonna a destra *)
	QuotaY_ColonnaSX : LREAL; 		(* Quota della colonna a destra *)
	QuotaAttualeAsse : LREAL; 		(* Quota attuale dell'asse Y*)
	QuotaDestinazioneAsse : LREAL; 	(* Quota Destinazione Asse Y*)
	IngombroOttimizzatoY_InTransito_Pos	: LREAL; (* Ingombro massimo della Y durante il ciclo in direzione POSITIVA *)
	IngombroOttimizzatoY_InTransito_Neg	: LREAL; (* Ingombro massimo della Y durante il ciclo in direzione NEGATIVA *)

	OffsetSicurezza_Y				: LREAL;  (* Offset sicurezza che si vuole mantenere dalle colonne *)
END_VAR
VAR_OUTPUT
	QuotaFuoriIngombro_Attuale_Y	: LREAL;
	QuotaFuoriIngombro_Destinazione_Y	: LREAL;
	//QuotaFuoriIngombro_Deposito_Y	: LREAL;
	Pinza_InIngombroColonne_Destinazione	: BOOL;
	Pinza_InIngombroColonne_Attuale			: BOOL;
END_VAR
VAR
	
END_VAR

(* Valutazione colonne in base al verso del pallettizzatore: verso stabilito guardando il pallettizzatore con la linea alle spalle *)
CASE VERSO_PALLETTIZZATORE OF
	PALLETTIZZATORE_DX:	// Colonna 6:DX, 5:SX
		(* Valuto la posizione attuale *)
		Pinza_InIngombroColonne_Attuale := FALSE;
		IF (QuotaAttualeAsse + IngombroOttimizzatoY_InTransito_Neg + OffsetSicurezza_Y <= QuotaY_ColonnaDX) THEN //Posizione Pinza - Metà ingombro - Offset sicurezza <= Ingombro colonna DX
			QuotaFuoriIngombro_Attuale_Y := QuotaY_ColonnaDX - IngombroOttimizzatoY_InTransito_Neg/2 - OffsetSicurezza_Y;
			Pinza_InIngombroColonne_Attuale := TRUE;
		END_IF
		IF (QuotaAttualeAsse - IngombroOttimizzatoY_InTransito_Pos - OffsetSicurezza_Y >= QuotaY_ColonnaSX) THEN //Posizione Pinza + Metà ingombro + Offset sicurezza >= Ingombro colonna SX
			QuotaFuoriIngombro_Attuale_Y := QuotaY_ColonnaSX + IngombroOttimizzatoY_InTransito_Pos/2 + OffsetSicurezza_Y;
			Pinza_InIngombroColonne_Attuale := TRUE;
		END_IF
		
		(* Valuto la posizione futura - Missione di Deposito/Prelievo *)
		Pinza_InIngombroColonne_Destinazione := FALSE;
		IF (QuotaDestinazioneAsse + IngombroOttimizzatoY_InTransito_Neg + OffsetSicurezza_Y <= QuotaY_ColonnaDX) THEN //Posizione Pinza - Metà ingombro - Offset sicurezza <= Ingombro colonna DX
			QuotaFuoriIngombro_Destinazione_Y := QuotaY_ColonnaDX - IngombroOttimizzatoY_InTransito_Neg - OffsetSicurezza_Y; 
			Pinza_InIngombroColonne_Destinazione := TRUE;
		END_IF
		IF (QuotaDestinazioneAsse - IngombroOttimizzatoY_InTransito_Pos - OffsetSicurezza_Y >= QuotaY_ColonnaSX) THEN //Posizione Pinza + Metà ingombro + Offset sicurezza >= Ingombro colonna SX
			QuotaFuoriIngombro_Destinazione_Y := QuotaY_ColonnaSX + IngombroOttimizzatoY_InTransito_Pos + OffsetSicurezza_Y;
			Pinza_InIngombroColonne_Destinazione := TRUE;
		END_IF
					
	PALLETTIZZATORE_SX: // Colonna 6:SX, 5:DX
		(* Valuto la posizione attuale *)
		Pinza_InIngombroColonne_Attuale := FALSE;
		IF (QuotaAttualeAsse + IngombroOttimizzatoY_InTransito_Pos + OffsetSicurezza_Y >= QuotaY_ColonnaDX) THEN //Posizione Pinza - Metà ingombro - Offset sicurezza <= Ingombro colonna 
			QuotaFuoriIngombro_Attuale_Y := QuotaY_ColonnaDX - IngombroOttimizzatoY_InTransito_Pos - OffsetSicurezza_Y;
			Pinza_InIngombroColonne_Attuale := TRUE;
		END_IF
		IF (QuotaAttualeAsse - IngombroOttimizzatoY_InTransito_Neg - OffsetSicurezza_Y <= QuotaY_ColonnaSX) THEN //Posizione Pinza + Metà ingombro + Offset sicurezza <= Ingombro colonna 
			QuotaFuoriIngombro_Attuale_Y := QuotaY_ColonnaSX + IngombroOttimizzatoY_InTransito_Neg + OffsetSicurezza_Y;
			Pinza_InIngombroColonne_Attuale := TRUE;
		END_IF
							
		(* Valuto la posizione futura - Missione di prelievo *)
		Pinza_InIngombroColonne_Destinazione := FALSE;
		IF (QuotaDestinazioneAsse + IngombroOttimizzatoY_InTransito_Pos + OffsetSicurezza_Y >= QuotaY_ColonnaDX) THEN //Posizione Pinza - Metà ingombro - Offset sicurezza <= Ingombro colonna 
			QuotaFuoriIngombro_Destinazione_Y := QuotaY_ColonnaDX - IngombroOttimizzatoY_InTransito_Pos - OffsetSicurezza_Y;
			Pinza_InIngombroColonne_Destinazione := TRUE;
		END_IF
		IF (QuotaDestinazioneAsse - IngombroOttimizzatoY_InTransito_Neg - OffsetSicurezza_Y <= QuotaY_ColonnaSX) THEN //Posizione Pinza + Metà ingombro + Offset sicurezza >= Ingombro colonna
			QuotaFuoriIngombro_Destinazione_Y := QuotaY_ColonnaSX + IngombroOttimizzatoY_InTransito_Neg + OffsetSicurezza_Y; 
			Pinza_InIngombroColonne_Destinazione := TRUE;
		END_IF

END_CASE

(* Nel caso in cui la pinza non sia in ingombro, fisso come fuori ingombro la quota attuale/ quota di destinazione dell'asse *)
IF NOT Pinza_InIngombroColonne_Attuale THEN
	QuotaFuoriIngombro_Attuale_Y := QuotaAttualeAsse;
END_IF
(* Nel caso in cui la pinza non sia in ingombro, fisso come fuori ingombro la quota di destinazione dell'asse *)
IF NOT Pinza_InIngombroColonne_Destinazione THEN
	QuotaFuoriIngombro_Destinazione_Y := QuotaAttualeAsse;
END_IF

END_FUNCTION_BLOCK

// ---- POUs/TFPalletizerDataTF/Utility Varie/TFCalcoloIngombroOttimizzatoPinza.TcPOU
FUNCTION_BLOCK TFCalcoloIngombroOttimizzatoPinza (* Calcola l'ingombro massimo assunto dalla pinza nelle direzioni X e Y durante il ciclo di lavoro *)
VAR_INPUT
	Quota_RotazioneAttuale : LREAL; //Angolo di rotazione attuale
	Quota_RotazioneDestinazione : LREAL;	//Angolo di rotazione destinazione
	IngombroSuperficialePinzaMAX : LREAL;	//Ingombro superficiale MASSIMO della pinza
	Larghezza : LREAL;	//Larghezza MASSIMA assunta dalla pinza
	Lunghezza: LREAL;	//Lunghezza MASSIMA assunta dall pinza
END_VAR
VAR_OUTPUT
	IngombroOttimizzatoY_InTransito : LREAL; //Ingombro MASSIMO in direzione Y
	IngombroOttimizzatoX_InTransito : LREAL; //Ingombro MASSIMO in direzione X
END_VAR
VAR
	Angolo : INT; //Angolo di appoggio per eseguire i calcoli
END_VAR

(* Fisso le quote al valore massimo *)
IngombroOttimizzatoY_InTransito := Dimensioni_Pinza.Lunghezza;
IngombroOttimizzatoX_InTransito := Dimensioni_Pinza.Lunghezza;
(* Fisso le quote al valore ottimale consideranto il valore massimo assunto durante tutta la rotazione della pinza durante il ciclo di lavoro *)
IF LREAL_TO_INT(Quota_RotazioneAttuale) <= LREAL_TO_INT(Quota_RotazioneDestinazione) THEN //Se l'angolo attuale di rotazione della pinza è INFERIORE alla posizione di destinazione
	FOR Angolo := LREAL_TO_INT(Quota_RotazioneAttuale) TO LREAL_TO_INT(Quota_RotazioneDestinazione) DO //Valuto tutti i gradi di rotazione in direzione CRESCENTE fino all'angolo di destinazione
		IF IngombroOttimizzatoX_InTransito < ABS(IngombroSuperficialePinzaMAX * SIN(deg_to_rad((ATAN(Larghezza/Lunghezza)*1/0.017+ Angolo)))) THEN
			IngombroOttimizzatoX_InTransito := ABS(IngombroSuperficialePinzaMAX * SIN(deg_to_rad((ATAN(Larghezza/Lunghezza)*1/0.017+ Angolo)))) ;
		END_IF
		IF IngombroOttimizzatoY_InTransito < ABS(IngombroSuperficialePinzaMAX * COS(deg_to_rad((ATAN(Larghezza/Lunghezza)*1/0.017+ Angolo)))) THEN
			IngombroOttimizzatoY_InTransito := ABS(IngombroSuperficialePinzaMAX * COS(deg_to_rad((ATAN(Larghezza/Lunghezza)*1/0.017+ Angolo))));
		END_IF
	END_FOR
	ELSIF LREAL_TO_INT(Quota_RotazioneAttuale) >= LREAL_TO_INT(Quota_RotazioneDestinazione) THEN //Se l'angolo attuale di rotazione della pinza è MAGGIORE alla posizione di destinazione
	FOR Angolo := LREAL_TO_INT(Quota_RotazioneAttuale) TO LREAL_TO_INT(Quota_RotazioneDestinazione) BY -1 DO //Valuto tutti i gradi di rotazione in direzione DECRESCENTE fino all'angolo di destinazione
		IF IngombroOttimizzatoX_InTransito < ABS(IngombroSuperficialePinzaMAX * SIN(deg_to_rad((ATAN(Larghezza/Lunghezza)*1/0.017+ Angolo)))) THEN
			IngombroOttimizzatoX_InTransito := ABS(IngombroSuperficialePinzaMAX * SIN(deg_to_rad((ATAN(Larghezza/Lunghezza)*1/0.017+ Angolo)))) ;
		END_IF
		IF IngombroOttimizzatoY_InTransito < ABS(IngombroSuperficialePinzaMAX * COS(deg_to_rad((ATAN(Larghezza/Lunghezza)*1/0.017+ Angolo)))) THEN
			IngombroOttimizzatoY_InTransito := ABS(IngombroSuperficialePinzaMAX * COS(deg_to_rad((ATAN(Larghezza/Lunghezza)*1/0.017+ Angolo))));
		END_IF
	END_FOR
END_IF

END_FUNCTION_BLOCK

// ---- POUs/TFPalletizerDataTF/Utility Varie/TFDirezioneAssePositiva.TcPOU
FUNCTION TFDirezioneAssePositiva : BOOL (*Valuta la direzione dell'asse in base alla sua quota attuale e alla sua destinazione*)
VAR_INPUT
	Posizione_Attuale 	: LREAL; //Posizione in cui si trova l'Asse
	Posizione_Finale 	: LREAL; //Posizione finale di posizionamento dell'Asse
END_VAR
VAR
END_VAR
(*Valuta la direzione dell'asse in base alla sua quota attuale e alla sua destinazione*)

TFDirezioneAssePositiva := FALSE;
IF Posizione_Attuale < Posizione_Finale THEN
	TFDirezioneAssePositiva := TRUE;
	RETURN;
END_IF

END_FUNCTION

// ---- POUs/TFPalletizerDataTF/TFPinzaInFuoriIngombroColonne_DirezioneX.TcPOU
(* Valuta se la pinza + il suo ingombro ha oltrepassato le colonne centrali *)
FUNCTION TFPinzaInFuoriIngombroColonne_DirezioneX : bool
VAR_INPUT
	DirezioneXPositiva : BOOL; //Indica che l'asse sta traslando in direzione Positiva
	AsseInMoto : BOOL; //Indica che lasse si sta muovento
	PosizioneAttuale : LREAL; //Posizione Attuale dell'asse
	IngombroX_Pos : LREAL; //Ingombro Attuale Pinza X Positivo
	IngombroX_Neg : LREAL; //Ingombro Attuale Pinza X Negativo
	PosizioneColonna_X : LREAL; //Posizione della colonna centrale in direzione X
	IngombroColonna_X : LREAL; //Ingobro della colonna in direzione X
END_VAR
VAR
END_VAR

TFPinzaInFuoriIngombroColonne_DirezioneX := FALSE;
(* Quota di Fuori-Ingombro della X rispetto le colonne, valutando l'ingombro effettivo della pinza *)
IF DirezioneXPositiva AND AsseInMoto THEN //Direzione POSITIVA con asse in moto
	IF (PosizioneAttuale - IngombroX_Neg)-50 >= (PosizioneColonna_X + IngombroColonna_X) THEN
		TFPinzaInFuoriIngombroColonne_DirezioneX := TRUE;
	END_IF
ELSIF NOT DirezioneXPositiva AND AsseInMoto THEN //Direzione NEGATIVA con asse in moto 
	IF (PosizioneAttuale + IngombroX_Pos)+50 < PosizioneColonna_X THEN
		TFPinzaInFuoriIngombroColonne_DirezioneX := TRUE;
	END_IF
ELSIF NOT AsseInMoto THEN //Se l'asse è fermo 
	IF (PosizioneAttuale - IngombroX_Neg)-50 >= (PosizioneColonna_X + IngombroColonna_X) OR // Se la quota attuale superiore alla posizione della colonna 
		(PosizioneAttuale + IngombroX_Pos)+50 < PosizioneColonna_X THEN 					// Se la quota attuale è inferiore alla posizione della colonna
			TFPinzaInFuoriIngombroColonne_DirezioneX := TRUE;
	END_IF
END_IF

END_FUNCTION

// ---- POUs/TFPalletizerDataTF/TFCalcoloPuntiDiAnticipoDinamici.TcPOU
FUNCTION_BLOCK TFCalcoloPuntiDiAnticipoDinamici
VAR_INPUT
	Traiettoria : POINTER TO TFTraiettoria;
	WorkSpace : POINTER TO TFMachinePalletizer_WorkSpace;
	WorkFootprint : POINTER TO ARRAY [1..MAXFOOTPRINT] OF TFMachinePalletizer_WorkFootprint; //Ingombri
	WorkPickPoint 				: POINTER TO ARRAY [1..MAXPICKPOINT] OF TFMachinePalletizer_WorkPickPointSlab;
	WorkPickPointState 			: POINTER TO ARRAY [1..MAXPICKPOINT] OF TFMachinePalletizer_WorkPickPoint_State;
	WorkPickPointOffset 		: POINTER TO ARRAY [1..MAXPICKPOINT] OF TFMachinePalletizer_WorkPickPointOffset;
	WorkPickPointDimension 		: POINTER TO ARRAY [1..MAXPICKPOINT] OF Work_PickPoint_Dimension;
	WorkArea : POINTER TO ARRAY [1..MAXAREA] OF TFMachinePalletizer_WorkArea;
	WorkAreaState : POINTER TO ARRAY [1..MAXAREA] OF TFMachinePalletizer_WorkAreaState;
	Pallet : POINTER TO ARRAY [1..MAXPALLET] OF TFMachinePalletizer_Pallet;
	Layer : POINTER TO ARRAY [1..MAXLAYER] OF TFMachinePalletizer_Layer;
	Forming : POINTER TO ARRAY [1..MAXFORMING] OF TFMachinePalletizer_FormingForSlab;
	PickPlaceParameters	: POINTER TO TFMachinePalletizer_ParametersFromHMI;
	Mission : POINTER TO TFMachinePalletizer_Mission;
	WorkAreaManager : POINTER TO TFWorkAreaManager;
	ModuleAX_X : POINTER TO TFModulePalletizer_Ax;
	ModuleAX_Y : POINTER TO TFModulePalletizer_Ax;
	ModuleAX_Z : POINTER TO TFModulePalletizer_Ax;
	ModuleAX_J : POINTER TO TFModulePalletizer_Ax;
	ModuleAX_K : POINTER TO TFModulePalletizer_Ax;
	AbilitaAnticipoDinamico : BOOL;
END_VAR
VAR
	f 		: INT;
	a 		: INT;
	P 		: UINT;
	wa 		: UINT;
	waDXSX 	: UINT;
	AltezzaDiIngombroArea 			: LREAL;
	AltezzaDiIngombroOstacoli 		: LREAL;
	AltezzaDiIngombroPuntiPrelievo 	: LREAL;
	AssegnaQuote 	: BOOL;
	
	LunghezzaMAX 	: LREAL;//LunghezzaMAX Totale pinza
	LarghezzaMAX 	: LREAL;//Larghezza Totale pinza
	SpessoreMAX  	: LREAL;//Spessore Totale pinza

	IngombroX_Pos 	: LREAL;//Ingombro della pinza nella Metà POSITIVA della pinza lungo X
	IngombroY_Pos 	: LREAL;//Ingombro della pinza nella Metà POSITIVA della pinza lungo Y
	IngombroZ_Pos 	: LREAL;//Ingombro della pinza nella Metà POSITIVA della pinza lungo Z
	
	IngombroX_Neg 	: LREAL;//Ingombro della pinza nella Metà NEGATIVA della pinza lungo X
	IngombroY_Neg 	: LREAL;//Ingombro della pinza nella Metà NEGATIVA della pinza lungo Y
	IngombroZ_Neg 	: LREAL;//Ingombro della pinza nella Metà NEGATIVA della pinza lungo Z
	
	IngombroY_Tot 	: LREAL;//Ingombro totale In direzione Y
	
	IngombroZ 	  : LREAL;//Ingombro della pinza lungo Z
	
	
	IngombroOttimizzatoX : LREAL;
	IngombroOttimizzatoY : LREAL;
	IngombroOttimizzatoZ : LREAL;

	IngombroVerticalePinzaMAX 		: LREAL;
	IngombroVerticaleMaxElementi 	: LREAL;
	
	DirezioneZPositiva : BOOL;
	DirezioneZNegativa : BOOL;
	
	WASX : UINT;
	WADX : UINT;
	WAPARTENZA : UINT;
	WADESTINAZIONE : UINT;
	LarghezzaPickPoint : REAL;
	TFCalcolaNumeroPostazioneDXSX : TFCalcolaNumeroPostazioneDXSX;
END_VAR

(* Calcolo gli ingombri della pinza nelle varie direzioni *)
(*TFCalcoliIngombroPinza(Mission := Mission,
						WorkAreaManager := WorkAreaManager,
						ModuleAX_X := ModuleAX_X,
						ModuleAX_Y := ModuleAX_Y,
						ModuleAX_Z := ModuleAX_Z,
						ModuleAX_J := ModuleAX_J,
						ModuleAX_K := ModuleAX_K,
						IngombroX_Pos := ADR(IngombroX_Pos),
						IngombroY_Pos := ADR(IngombroY_Pos),
						IngombroX_Neg := ADR(IngombroX_Neg),
						IngombroY_Neg := ADR(IngombroY_Neg),
						IngombroY_Tot := ADR(IngombroY_Tot),
						IngombroZ_Pos := ADR(IngombroZ_Pos),
						IngombroZ_Neg := ADR(IngombroZ_Neg));
		*)										
////////////////////////////////////////////////////////////////////////////////////////////////////////////////////////////////////////////////////////////
///////////////////////////////////////////////////////////////////////////////////////////////////////////////////////////////////////////////////////////

(* Larhezza Pick Point + Pacco *)
(*IF WorkPickPointState^[1].XDim >= WorkPickPointDimension[1].XDim THEN
	LarghezzaPickPoint := WorkPickPointState^[1].XDim;
else
	LarghezzaPickPoint := WorkPickPointDimension[1].Xdim;
END_IF
*)
(*************************** Anticipo asse X *************************************)
QuotaAnticipoDinamicaX_Raggiunta := FALSE; 

(*************************** Anticipo dell'asse Z *********************************) 
(* Valuto la direzione della Z *)
DirezioneZPositiva := TFDirezioneAssePositiva(Posizione_Attuale:=ModuleAX_Z^.Ax^.Status.ActPosition,Posizione_Finale:=Mission^.ZPick);
DirezioneZNegativa := NOT DirezioneZPositiva;

IngombroVerticaleMaxElementi := 0;

(* Anticipo Y per Deposito Pacco *)
QuotaAnticipoDinamicaY_Raggiunta := FALSE;

(*
	IF Mission^.PPick = INT_TO_UINT(TPICK_PACK) AND Mission^.State = MISSION_STATE_DEPOSITO_PACCO_RUN  THEN
		IF (Mission^.YPlace >= Mission^.YPick) THEN //Se deposito un pacco orrizzontale e la posizione di deposito super la posizione Y di prelievo
			QuotaAnticipoDinamicaY_Raggiunta := TRUE;
		ELSE
			QuotaAnticipoDinamicaY_Raggiunta := FALSE;
		END_IF
	ELSE
		QuotaAnticipoDinamicaY_Raggiunta := FALSE;
	END_IF*)
	
